# B&R Automation Studio project DeltaTracking
Automation Studio 6.3.0.261; technology packages: mappCockpit 6.0.0, mappMotion 6.4.0, mappView 6.0.0, OpcUaCs 6.0.0

## Configuration Config1

CPU 5APC3100.KBU3-000, AutomationRuntime 6.4.0, Build 11.3.0, Safety 0.0, Vc 

### Task classes (Cpu.sw)
```
Cyclic#1 (cycle 2000 us, tolerance 0 us):
  APP_Convey <- Conveyor.APP_Conveyor1.prg
  APP_Conve1 <- Conveyor.APP_Conveyor2.prg
  APP_Robot1 <- Robots.Robot1.APP_Robot1.prg
DataObjects: Arnc0sys, Acp10sys
NcDataObjects: gmcipuc, gmciplog, gmcipfub, gmcipfun, gmciplsm, gmciplbr, gmcipmxd, gmcipvar, gmcipsys, gmcipiec, gmcipesm, gmcipusm, gmcipcsm, gmcipui, gmcipubr, gmcipcbr, gmcipcfg, gmcipus, gmcipmx, Cam
Binaries: McAcpSys, mcdrivelog, udbdef, TCData, mvLoader, arsvcreg, arflatprv, mCoWebSc, McAcpDrv, McAcpSim, McProfGen, McMechSys, arcoal, ashwac, arconfig, asfw, ashwd, iomap, User, Role, sysconf, TraceConfi, Settings, Config_1, Hierarchy, Config, AxisAx_1, Config_2, ComRobot, Config_4, Config_5, Config_3, Config_6, ToolX20, AxesAxX21, GRobot1, GFRobot1, ARobot1, ComRobot1, WorkRobot1, GRobot2, MRobot1, GFRobot2, FeatX21, TrkDevX21, TrkDevConv, AxisAxX25, MecX20, AxesAxX20, WorkX20, FeatX20, DeltaX20, ComFeatX20, DeltaX21, TrkDevX20, vccddbox, vcfile, vccbtn, vcpdvnc, arialbd, vcmgr, vctcal, vcgclass, vcctext, vccnum, vcfntttf, vcdsloc, vccstr, arial, Visu03, vccshape, vcalarm, Visu01, vccdt, vccscale, vcchtml, vcchspot, vccbmp, vccpopup, vcshared, vcxml, vccurl, vcrt, vccslider, Visu02, vcnet, vcclbox, vcbclass, vcdsint, vcpdsw, vccovl, vccline, TCLang, visvc, vccdbox, vcpfar00, vcpfmtcx, vcpfapc, GrpMaster, Users, UsersLogin, TC, Files, DiagWebXs, AlmMaster, AlmHisMain, AlmMain, GrpVMaster, AlmVMaster, CfgPureVir, AxisPS, AxisAxXX1, AxisAxXX2, AxisMaster, MDevXX1, AxVMaster, GrpDevXX1, AlmDevXX1, GrPDevXX4, AlmDevXX4, GrPDevX10, AlmDevX10, AlmDevX20, GrpDevX20, AlmDevX21, GrpDevX21, AlmMBelts, GrpMBelts, AlmDevXX6, GrpDevXX6, AxesVAxX20, vcpfx20, AxisMBelts, MasMBelts, MBeltsPt, AxesVAxX25, AxesAxX10, AxesAxX25, WorkX10, CncXX6, MecX10, AxesVAxX10, DeltaX10, FeatXX6, FeatX10, ToolX10, ToolXX6, MecXX6, MotMaster, MotVMaster, vcctrend, MotDevX10, GrPDevXX3, AlmDevXX3, MotDevXX3, GrPDevXX2, MotDevXX1, AlmDevXX2, MotDevXX2, vcpkat, arnc0cfg, Sdc10map, Arnc0map, Sdc10map1, Sdc10map2, MotDevX20, MotDevX11, MotDevXX9, GrpDevXX9, AlmDevXX9, PML, MotDevXX6, CncDevXX6, MotDevXX7, AlmDevXX7, GrpDevXX7, Robot, AlmDevXX8, GrpDevXX8, MotSim, MotSpindle, MotDevXXA, AlmDevXXA, GrpDevXXA, GrpDevX11, AlmDevX11, OpcUaBasic, User_1, OpcUaMap, AlmHmi, AlmHistHmi, Groups, vccpiech, MotMac, acp10cfg, Acp10map
Libraries: standard, AsBrStr, sys_lib, runtime, AsArSdm, astime, brsystem, FileIO, AsIODiag, DataObj, AsArProf, AsMem, AsIOAcc, AsEPL, ASMcDcs, AsBrMath, visapi, ArTextSys, AsSem, AsIecCon, AsZip, MpRecipe, MpUserX, MpFile, MpAlarmX, MpCom, CoTrace, MpServer, powerlnk, aruser, asusb, ashw, arcert, arssl, aseth, asio, vcresman, IecCheck, areventlog, MpBase, McBase, McAxGroup, McAcpAx, McAxis, McPathGen, McTrkPath, MpAxis, McProgInt, McPureVAx, McDS402Ax, MpRobotics, MpCnc
```

### Hardware
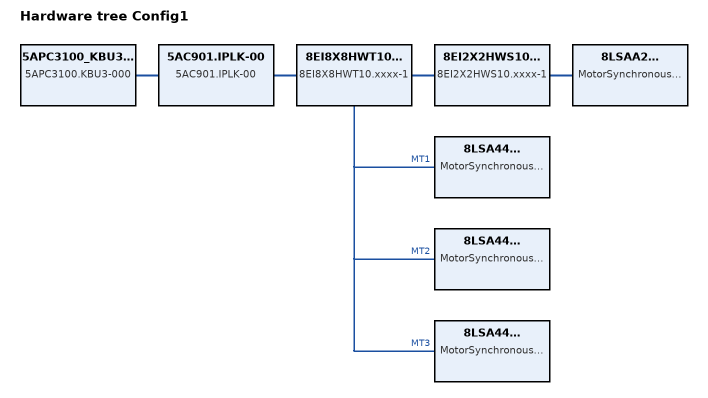
```
5AC901.IPLK-00 : 5AC901.IPLK-00 v2.0.0.0  [SL -> 5APC3100_KBU3_000.SL2]
  Connector IF1:
    DNAConfiguration = manual
    Channel1
    ChannelID1 = McAcpBroadcast
    ChannelType1 = OCTET[96]
5APC3100_KBU3_000 : 5APC3100.KBU3-000 v2.2.7.0
  Connector IF3:
    AssignedOperatingSystem = ARemb
    ActivateDevice = 1
    HostName = apc3100robert
    Mode = Manual
    InternetAddress = 10.43.51.43
    SubnetMask = 255.255.255.0
    Vnc1
    VncKeyMappingFile1 = 
    VncRefreshRate1 = 100
    ActivateSnmp = 2
  Connector IF4:
    AssignedOperatingSystem = ARemb
    ActivateDevice = 1
    HostName = apc3100robert
    Mode = DHCPServer
    InternetAddress = 192.168.20.254
    SubnetMask = 255.255.255.0
    Lease1
    LeaseName1 = Range1
    LeaseStartAddress1 = 192.168.20.100
    LeaseStopAddress1 = 192.168.20.110
    LeaseSubnetMask1 = 255.255.255.0
    Vnc1
    VncTitle1 = VNC
    ActivateSnmp = 2
  Connector IF5:
    AssignedOperatingSystem = ARemb
  Connector IF6:
    AssignedOperatingSystem = ARemb
  Connector IF7:
    AssignedOperatingSystem = ARemb
  Connector IF8:
    AssignedOperatingSystem = ARemb
  ConfigurationID = Template_X20CP1586
  UserPartitionSize = 5
  Simulation = 1
  TimerDeviceType = EPLX2X
  TimerDevice = 5AC901.IPLK-00.IF1
  IdleTaskClass = 4
  TaskClassIdleTime = 4000
  Cyclic1Duration = 2000
  Cyclic1Tolerance = 0
  Cyclic1Stack = 16384
  Cyclic2Duration = 4000
  Cyclic2Tolerance = 0
  Cyclic3Duration = 10000
  Cyclic3Tolerance = 0
  Cyclic4Duration = 20000
  Cyclic4Tolerance = 0
  Cyclic5Duration = 50000
  Cyclic5Tolerance = 0
  Cyclic6Duration = 100000
  Cyclic6Tolerance = 0
  Cyclic7Duration = 200000
  Cyclic7Tolerance = 0
  FileDevice1
  FileDeviceName1 = SceneViewer
  FileDevicePath1 = USER_PATH
  FileDevice2
  FileDeviceName2 = MPLogDir
  FileDevicePath2 = USER_PATH\Log
  FileDevice3
  FileDeviceName3 = DebugData
  FileDevicePath3 = USER_PATH\\Debug
  FileDevice4
  FileDeviceName4 = CNC_Prg
  FileDevicePath4 = USER_PATH\CNC_Prg
  EthernetDefaultGateway = 10.43.51.1
  ActivateFtpServer = 1
  FTPProtocol = 2
  FtpUser1
  FtpUsername1 = gmctest
  FtpUserPassword1 = dJg12F/7hd2fGO/QauVo5qNTeUud8LRwkPqca2btE1Q=
  FtpUserSalt1 = iGhlfz5v
  FTPAccessRight1 = 0
  FTPdevice1 = ALL
  ActivateWebServer = 1
  ActivateSdm = 1
8EI2X2HWS10.xxxx-1-QC_D4r1100R_1 : 8EI2X2HWS10.xxxx-1 v2.4.0.0 (NodeNumber=6)  [PLK1 -> 8EI8X8HWT10.xxxx-1-Q1-Q2-Q3_D4r1100R_1.PLK2 [Cable Type=PowerlinkCable, Length=10, Version=1.0.0.3]]
  DriveConfiguration/Encoder/EncoderX41:
    InterfaceType = EnDat
  DriveConfiguration/Channel[1]/RealAxis:
    AxisReference = gAxisQC_D4r1100R_1
  DriveConfiguration/Channel[1]/RealAxis/MechanicalElements/Gearbox:
    InputIsReadOnly = 1
    Input = 10
    OutputIsReadOnly = 1
  DriveConfiguration/Channel[1]/RealAxis/MechanicalElements/RotaryToLinearTransformation:
    ReferenceDistanceIsReadOnly = 1
    ReferenceDistance = 360
  DriveConfiguration/Channel[1]/RealAxis/Controller:
    ModeIsReadOnly = 1
    Mode = PositionControllerWithTorqueFeedForward
  DriveConfiguration/Channel[1]/RealAxis/Controller/Mode/Position:
    ProportionalGainIsReadOnly = 1
    ProportionalGain = 80.0
    IntegrationTimeIsReadOnly = 1
  DriveConfiguration/Channel[1]/RealAxis/Controller/Mode/Speed:
    ProportionalGainIsReadOnly = 1
    IntegrationTimeIsReadOnly = 1
    FilterTimeIsReadOnly = 1
  DriveConfiguration/Channel[1]/RealAxis/Controller/Mode:
    FeedForwardIsReadOnly = 1
    FeedForward = CyclicValueFromAxesGroup
  DriveConfiguration/Channel[1]/RealAxis/Controller/Mode/LoopFilters:
    LoopFilterXIsReadOnly = 1
  DriveConfiguration/Channel[1]/RealAxis/Homing:
    Mode = Absolute
    RestorePositionVariable = 
  DriveConfiguration/Channel[1]/RealAxis/StopReaction:
    DriveError = CyclicDecelerationFromAxesGroup
  DriveConfiguration/Channel[1]/RealAxis/MovementErrorLimits:
    PositionError = 0.5
  DriveConfiguration/Channel[1]/RealAxis:
    JerkFilterIsReadOnly = 1
    JerkFilter = Used
  DriveConfiguration/Channel[1]/RealAxis/JerkFilter:
    JerkTimeMin = 0.06
    JerkTime = 0.06
8EI8X8HWT10.xxxx-1-Q1-Q2-Q3_D4r1100R_1 : 8EI8X8HWT10.xxxx-1 v2.4.0.0 (NodeNumber=4)  [PLK1 -> 5AC901.IPLK-00.IF1 [Cable Type=PowerlinkCable, Length=10, Version=1.0.0.3]; PLK2 -> 8EI2X2HWS10.xxxx-1-QC_D4r1100R_1.PLK1 [Cable Type=PowerlinkCable, Length=10, Version=1.0.0.3]; MT2 -> 8LSA44.DB060S200-3_Q2_D4r1100R_1.MT; MT3 -> 8LSA44.DB060S200-3_Q3_D4r1100R_1.MT]
  DriveConfiguration/Encoder/EncoderX41:
    InterfaceType = EnDat
  DriveConfiguration/Encoder/EncoderX42:
    InterfaceType = EnDat
  DriveConfiguration/Encoder/EncoderX43:
    InterfaceType = EnDat
  DriveConfiguration/Channel[1]/RealAxis:
    AxisReference = gAxisQ1_D4r1100R_1
  DriveConfiguration/Channel[1]/RealAxis/MechanicalElements/Gearbox:
    InputIsReadOnly = 1
    Input = 28
    OutputIsReadOnly = 1
  DriveConfiguration/Channel[1]/RealAxis/MechanicalElements/RotaryToLinearTransformation:
    ReferenceDistanceIsReadOnly = 1
    ReferenceDistance = 360
  DriveConfiguration/Channel[1]/RealAxis/Controller:
    ModeIsReadOnly = 1
    Mode = PositionControllerWithTorqueFeedForward
  DriveConfiguration/Channel[1]/RealAxis/Controller/Mode/Position:
    ProportionalGainIsReadOnly = 1
    ProportionalGain = 150.0
    IntegrationTimeIsReadOnly = 1
  DriveConfiguration/Channel[1]/RealAxis/Controller/Mode/Speed:
    ProportionalGainIsReadOnly = 1
    ProportionalGain = 7.5
    IntegrationTimeIsReadOnly = 1
    FilterTimeIsReadOnly = 1
  DriveConfiguration/Channel[1]/RealAxis/Controller/Mode:
    FeedForwardIsReadOnly = 1
    FeedForward = CyclicValueFromAxesGroup
  DriveConfiguration/Channel[1]/RealAxis/Controller/Mode/LoopFilters:
    LoopFilterXIsReadOnly = 1
  DriveConfiguration/Channel[1]/RealAxis/Homing:
    Mode = Absolute
    RestorePositionVariable = 
  DriveConfiguration/Channel[1]/RealAxis/StopReaction:
    DriveError = CyclicDecelerationFromAxesGroup
  DriveConfiguration/Channel[1]/RealAxis/MovementErrorLimits:
    PositionError = 0.5
  DriveConfiguration/Channel[1]/RealAxis:
    JerkFilterIsReadOnly = 1
    JerkFilter = Used
  DriveConfiguration/Channel[1]/RealAxis/JerkFilter:
    JerkTimeMin = 0.06
    JerkTime = 0.06
  DriveConfiguration/Channel[2]/RealAxis:
    AxisReference = gAxisQ2_D4r1100R_1
  DriveConfiguration/Channel[2]/RealAxis/MechanicalElements/Gearbox:
    InputIsReadOnly = 1
    Input = 28
    OutputIsReadOnly = 1
  DriveConfiguration/Channel[2]/RealAxis/MechanicalElements/RotaryToLinearTransformation:
    ReferenceDistanceIsReadOnly = 1
    ReferenceDistance = 360
  DriveConfiguration/Channel[2]/RealAxis/Controller:
    ModeIsReadOnly = 1
    Mode = PositionControllerWithTorqueFeedForward
  DriveConfiguration/Channel[2]/RealAxis/Controller/Mode/Position:
    ProportionalGainIsReadOnly = 1
    ProportionalGain = 150.0
    IntegrationTimeIsReadOnly = 1
  DriveConfiguration/Channel[2]/RealAxis/Controller/Mode/Speed:
    ProportionalGainIsReadOnly = 1
    ProportionalGain = 7.5
    IntegrationTimeIsReadOnly = 1
    FilterTimeIsReadOnly = 1
  DriveConfiguration/Channel[2]/RealAxis/Controller/Mode:
    FeedForwardIsReadOnly = 1
    FeedForward = CyclicValueFromAxesGroup
  DriveConfiguration/Channel[2]/RealAxis/Controller/Mode/LoopFilters:
    LoopFilterXIsReadOnly = 1
  DriveConfiguration/Channel[2]/RealAxis/Homing:
    Mode = Absolute
    RestorePositionVariable = 
  DriveConfiguration/Channel[2]/RealAxis/StopReaction:
    DriveError = CyclicDecelerationFromAxesGroup
  DriveConfiguration/Channel[2]/RealAxis/MovementErrorLimits:
    PositionError = 0.5
  DriveConfiguration/Channel[2]/RealAxis:
    JerkFilterIsReadOnly = 1
    JerkFilter = Used
  DriveConfiguration/Channel[2]/RealAxis/JerkFilter:
    JerkTimeMin = 0.06
    JerkTime = 0.06
  DriveConfiguration/Channel[3]/RealAxis:
    AxisReference = gAxisQ3_D4r1100R_1
  DriveConfiguration/Channel[3]/RealAxis/MechanicalElements/Gearbox:
    InputIsReadOnly = 1
    Input = 28
    OutputIsReadOnly = 1
  DriveConfiguration/Channel[3]/RealAxis/MechanicalElements/RotaryToLinearTransformation:
    ReferenceDistanceIsReadOnly = 1
    ReferenceDistance = 360
  DriveConfiguration/Channel[3]/RealAxis/Controller:
    ModeIsReadOnly = 1
    Mode = PositionControllerWithTorqueFeedForward
  DriveConfiguration/Channel[3]/RealAxis/Controller/Mode/Position:
    ProportionalGainIsReadOnly = 1
    ProportionalGain = 150.0
    IntegrationTimeIsReadOnly = 1
  DriveConfiguration/Channel[3]/RealAxis/Controller/Mode/Speed:
    ProportionalGainIsReadOnly = 1
    ProportionalGain = 7.5
    IntegrationTimeIsReadOnly = 1
    FilterTimeIsReadOnly = 1
  DriveConfiguration/Channel[3]/RealAxis/Controller/Mode:
    FeedForwardIsReadOnly = 1
    FeedForward = CyclicValueFromAxesGroup
  DriveConfiguration/Channel[3]/RealAxis/Controller/Mode/LoopFilters:
    LoopFilterXIsReadOnly = 1
  DriveConfiguration/Channel[3]/RealAxis/Homing:
    Mode = Absolute
    RestorePositionVariable = 
  DriveConfiguration/Channel[3]/RealAxis/StopReaction:
    DriveError = CyclicDecelerationFromAxesGroup
  DriveConfiguration/Channel[3]/RealAxis/MovementErrorLimits:
    PositionError = 0.5
  DriveConfiguration/Channel[3]/RealAxis:
    JerkFilterIsReadOnly = 1
    JerkFilter = Used
  DriveConfiguration/Channel[3]/RealAxis/JerkFilter:
    JerkTimeMin = 0.06
    JerkTime = 0.06
8LSA44.DB060S200-3_Q1_D4r1100R_1 : MotorSynchronous_any v2.2.1.0  [MT -> 8EI8X8HWT10.xxxx-1-Q1-Q2-Q3_D4r1100R_1.MT1]
  M1/MotorParameters:
    MOTOR_POLEPAIRS = 5
    MOTOR_SPEED_RATED = 6000
    MOTOR_SPEED_MAX = 12000
    MOTOR_VOLTAGE_RATED = 400
    MOTOR_CURR_RATED = 3.7
    MOTOR_CURR_STALL = 7.4
    MOTOR_CURR_MAX = 43.8
    MOTOR_TORQ_RATED = 3
    MOTOR_TORQ_STALL = 6
    MOTOR_TORQ_MAX = 22.8
    MOTOR_VOLTAGE_CONST = 49.22
    MOTOR_TORQ_CONST = 0.81
    MOTOR_STATOR_RESISTANCE = 0.863
    MOTOR_STATOR_INDUCTANCE = 6.2
    MOTOR_INERTIA = 2.73
    VoltageLimitation = Used
  M1/MotorParameters/VoltageLimitation:
    MOTOR_UDC_MAX = 1000
  M1/MotorParameters/EncoderMounting:
    Angle = StoredOnEncoder
  M1/MotorParameters/TemperatureSensor:
    MOTOR_TEMPSENS_LIM = 130
    TemperatureSensorInterface = EncoderConnectorDigital
    MOTOR_TEMPSENS_PAR1 = 30
    MOTOR_TEMPSENS_PAR2 = 254
    MOTOR_TEMPSENS_PAR3 = -29.72
    MOTOR_TEMPSENS_PAR4 = -4.58
    MOTOR_TEMPSENS_PAR5 = 20.33
    MOTOR_TEMPSENS_PAR6 = 45.18
    MOTOR_TEMPSENS_PAR7 = 69.96
    MOTOR_TEMPSENS_PAR8 = 94.71
    MOTOR_TEMPSENS_PAR9 = 119.6
    MOTOR_TEMPSENS_PAR10 = 149.11
  M1/MotorParameters/TemperatureModel:
    MOTOR_WIND_TEMP_MAX = 110
  M1/MotorParameters/TemperatureModel/Calculation:
    MOTOR_WIND_CROSS_SECT = 0.985
    MOTOR_TAU_THERM = 1800
  M1:
    Brake = Used
  M1/Brake:
    MOTOR_BRAKE_CURR_RATED = 0.83
    MOTOR_BRAKE_TORQ_RATED = 8
    MOTOR_BRAKE_ON_TIME = 0.038
    MOTOR_BRAKE_OFF_TIME = 0.055
    MOTOR_BRAKE_INERTIA = 0.69
  M1/Encoder:
    MOTOR_ENCOD_ATTR = 1
    MOTOR_ENCOD_INERTIA = 0.022
    TemperatureSensor = Used
  M1/Encoder/TemperatureSensor:
    MOTOR_ENCOD_TEMP_LIM = 129
  M1:
    Gearbox = UsedWithDynamicTorqueLimitation
  M1/Gearbox/GearRatio:
    Input = 28
  M1/Gearbox:
    MOTORGEAR_SPEED_MAX = 7500
    MOTORGEAR_TORQ_NOM = 126
    MOTORGEAR_TORQ_MAX = 126
    MOTORGEAR_INERTIA = 0.51
    MOTORGEAR_VISC_FRIC = 0.002
    MOTORGEAR_STAT_FRIC = 0.22
8LSA44.DB060S200-3_Q2_D4r1100R_1 : MotorSynchronous_any v2.2.1.0  [MT -> 8EI8X8HWT10.xxxx-1-Q1-Q2-Q3_D4r1100R_1.MT2]
  M1/MotorParameters:
    MOTOR_POLEPAIRS = 5
    MOTOR_SPEED_RATED = 6000
    MOTOR_SPEED_MAX = 12000
    MOTOR_VOLTAGE_RATED = 400
    MOTOR_CURR_RATED = 3.7
    MOTOR_CURR_STALL = 7.4
    MOTOR_CURR_MAX = 43.8
    MOTOR_TORQ_RATED = 3
    MOTOR_TORQ_STALL = 6
    MOTOR_TORQ_MAX = 22.8
    MOTOR_VOLTAGE_CONST = 49.22
    MOTOR_TORQ_CONST = 0.81
    MOTOR_STATOR_RESISTANCE = 0.863
    MOTOR_STATOR_INDUCTANCE = 6.2
    MOTOR_INERTIA = 2.73
    VoltageLimitation = Used
  M1/MotorParameters/VoltageLimitation:
    MOTOR_UDC_MAX = 1000
  M1/MotorParameters/EncoderMounting:
    Angle = StoredOnEncoder
  M1/MotorParameters/TemperatureSensor:
    MOTOR_TEMPSENS_LIM = 130
    TemperatureSensorInterface = EncoderConnectorDigital
    MOTOR_TEMPSENS_PAR1 = 30
    MOTOR_TEMPSENS_PAR2 = 254
    MOTOR_TEMPSENS_PAR3 = -29.72
    MOTOR_TEMPSENS_PAR4 = -4.58
    MOTOR_TEMPSENS_PAR5 = 20.33
    MOTOR_TEMPSENS_PAR6 = 45.18
    MOTOR_TEMPSENS_PAR7 = 69.96
    MOTOR_TEMPSENS_PAR8 = 94.71
    MOTOR_TEMPSENS_PAR9 = 119.6
    MOTOR_TEMPSENS_PAR10 = 149.11
  M1/MotorParameters/TemperatureModel:
    MOTOR_WIND_TEMP_MAX = 110
  M1/MotorParameters/TemperatureModel/Calculation:
    MOTOR_WIND_CROSS_SECT = 0.985
    MOTOR_TAU_THERM = 1800
  M1:
    Brake = Used
  M1/Brake:
    MOTOR_BRAKE_CURR_RATED = 0.83
    MOTOR_BRAKE_TORQ_RATED = 8
    MOTOR_BRAKE_ON_TIME = 0.038
    MOTOR_BRAKE_OFF_TIME = 0.055
    MOTOR_BRAKE_INERTIA = 0.69
  M1/Encoder:
    MOTOR_ENCOD_ATTR = 1
    MOTOR_ENCOD_INERTIA = 0.022
    TemperatureSensor = Used
  M1/Encoder/TemperatureSensor:
    MOTOR_ENCOD_TEMP_LIM = 129
  M1:
    Gearbox = UsedWithDynamicTorqueLimitation
  M1/Gearbox/GearRatio:
    Input = 28
  M1/Gearbox:
    MOTORGEAR_SPEED_MAX = 7500
    MOTORGEAR_TORQ_NOM = 126
    MOTORGEAR_TORQ_MAX = 126
    MOTORGEAR_INERTIA = 0.51
    MOTORGEAR_VISC_FRIC = 0.002
    MOTORGEAR_STAT_FRIC = 0.22
8LSA44.DB060S200-3_Q3_D4r1100R_1 : MotorSynchronous_any v2.2.1.0  [MT -> 8EI8X8HWT10.xxxx-1-Q1-Q2-Q3_D4r1100R_1.MT3]
  M1/MotorParameters:
    MOTOR_POLEPAIRS = 5
    MOTOR_SPEED_RATED = 6000
    MOTOR_SPEED_MAX = 12000
    MOTOR_VOLTAGE_RATED = 400
    MOTOR_CURR_RATED = 3.7
    MOTOR_CURR_STALL = 7.4
    MOTOR_CURR_MAX = 43.8
    MOTOR_TORQ_RATED = 3
    MOTOR_TORQ_STALL = 6
    MOTOR_TORQ_MAX = 22.8
    MOTOR_VOLTAGE_CONST = 49.22
    MOTOR_TORQ_CONST = 0.81
    MOTOR_STATOR_RESISTANCE = 0.863
    MOTOR_STATOR_INDUCTANCE = 6.2
    MOTOR_INERTIA = 2.73
    VoltageLimitation = Used
  M1/MotorParameters/VoltageLimitation:
    MOTOR_UDC_MAX = 1000
  M1/MotorParameters/EncoderMounting:
    Angle = StoredOnEncoder
  M1/MotorParameters/TemperatureSensor:
    MOTOR_TEMPSENS_LIM = 130
    TemperatureSensorInterface = EncoderConnectorDigital
    MOTOR_TEMPSENS_PAR1 = 30
    MOTOR_TEMPSENS_PAR2 = 254
    MOTOR_TEMPSENS_PAR3 = -29.72
    MOTOR_TEMPSENS_PAR4 = -4.58
    MOTOR_TEMPSENS_PAR5 = 20.33
    MOTOR_TEMPSENS_PAR6 = 45.18
    MOTOR_TEMPSENS_PAR7 = 69.96
    MOTOR_TEMPSENS_PAR8 = 94.71
    MOTOR_TEMPSENS_PAR9 = 119.6
    MOTOR_TEMPSENS_PAR10 = 149.11
  M1/MotorParameters/TemperatureModel:
    MOTOR_WIND_TEMP_MAX = 110
  M1/MotorParameters/TemperatureModel/Calculation:
    MOTOR_WIND_CROSS_SECT = 0.985
    MOTOR_TAU_THERM = 1800
  M1:
    Brake = Used
  M1/Brake:
    MOTOR_BRAKE_CURR_RATED = 0.83
    MOTOR_BRAKE_TORQ_RATED = 8
    MOTOR_BRAKE_ON_TIME = 0.038
    MOTOR_BRAKE_OFF_TIME = 0.055
    MOTOR_BRAKE_INERTIA = 0.69
  M1/Encoder:
    MOTOR_ENCOD_ATTR = 1
    MOTOR_ENCOD_INERTIA = 0.022
    TemperatureSensor = Used
  M1/Encoder/TemperatureSensor:
    MOTOR_ENCOD_TEMP_LIM = 129
  M1:
    Gearbox = UsedWithDynamicTorqueLimitation
  M1/Gearbox/GearRatio:
    Input = 28
  M1/Gearbox:
    MOTORGEAR_SPEED_MAX = 7500
    MOTORGEAR_TORQ_NOM = 126
    MOTORGEAR_TORQ_MAX = 126
    MOTORGEAR_INERTIA = 0.51
    MOTORGEAR_VISC_FRIC = 0.002
    MOTORGEAR_STAT_FRIC = 0.22
8LSAA2.D9045S200-3_QC_D4r1100R_1 : MotorSynchronous_any v2.2.1.0  [MT -> 8EI2X2HWS10.xxxx-1-QC_D4r1100R_1.MT1]
  M1/MotorParameters:
    MOTOR_POLEPAIRS = 5
    MOTOR_SPEED_RATED = 4500
    MOTOR_SPEED_MAX = 7000
    MOTOR_VOLTAGE_RATED = 400
    MOTOR_CURR_RATED = 1.31
    MOTOR_CURR_STALL = 1.42
    MOTOR_CURR_MAX = 6
    MOTOR_TORQ_RATED = 1.27
    MOTOR_TORQ_STALL = 1.4
    MOTOR_TORQ_MAX = 4.5
    MOTOR_VOLTAGE_CONST = 58.64
    MOTOR_TORQ_CONST = 0.97
    MOTOR_STATOR_RESISTANCE = 13.9
    MOTOR_STATOR_INDUCTANCE = 27
    MOTOR_INERTIA = 0.38
    VoltageLimitation = Used
  M1/MotorParameters/VoltageLimitation:
    MOTOR_UDC_MAX = 1000
  M1/MotorParameters/EncoderMounting:
    Angle = StoredOnEncoder
  M1/MotorParameters/TemperatureSensor:
    MOTOR_TEMPSENS_LIM = 130
    TemperatureSensorInterface = EncoderConnectorDigital
    MOTOR_TEMPSENS_PAR1 = 30
    MOTOR_TEMPSENS_PAR2 = 254
    MOTOR_TEMPSENS_PAR3 = -29.72
    MOTOR_TEMPSENS_PAR4 = -4.58
    MOTOR_TEMPSENS_PAR5 = 20.33
    MOTOR_TEMPSENS_PAR6 = 45.18
    MOTOR_TEMPSENS_PAR7 = 69.96
    MOTOR_TEMPSENS_PAR8 = 94.71
    MOTOR_TEMPSENS_PAR9 = 119.6
    MOTOR_TEMPSENS_PAR10 = 149.11
  M1/MotorParameters/TemperatureModel:
    MOTOR_WIND_TEMP_MAX = 110
  M1/MotorParameters/TemperatureModel/Calculation:
    MOTOR_WIND_CROSS_SECT = 0.126
    MOTOR_TAU_THERM = 1860
  M1:
    Brake = Used
  M1/Brake:
    MOTOR_BRAKE_CURR_RATED = 0.56
    MOTOR_BRAKE_TORQ_RATED = 3.2
    MOTOR_BRAKE_ON_TIME = 0.01
    MOTOR_BRAKE_OFF_TIME = 0.06
    MOTOR_BRAKE_INERTIA = 0.38
  M1/Encoder:
    MOTOR_ENCOD_ATTR = 1
    MOTOR_ENCOD_INERTIA = 0.004
    TemperatureSensor = Used
  M1/Encoder/TemperatureSensor:
    MOTOR_ENCOD_TEMP_LIM = 124
  M1:
    Gearbox = UsedWithDynamicTorqueLimitation
  M1/Gearbox/GearRatio:
    Input = 10
  M1/Gearbox:
    MOTORGEAR_SPEED_MAX = 7500
    MOTORGEAR_TORQ_NOM = 7.0
    MOTORGEAR_TORQ_MAX = 7.0
    MOTORGEAR_INERTIA = 0.16
    MOTORGEAR_VISC_FRIC = 0.0038
    MOTORGEAR_STAT_FRIC = 0.07
```

### Config_11.axesgroupfeature - 5APC3100_KBU3_000/mappMotion/Codian_D4r1100R_1/Config_11.axesgroupfeature
```
Element Feature_Programs_D4r1100R_1 (Type=axesgroupfeature)
  Type:
    InitialSettings:
      AccuracyHoldDelays = User defined
        UserAxesDelay = 0.03
    Location = User
      UserLocation[1]:
        FileDevice = CNC_Prg
```

### Config_2.axesgroup - 5APC3100_KBU3_000/mappMotion/Codian_D4r1100R_1/Config_2.axesgroup
```
Element gAxesGroup_D4r1100R_1 (Type=axesgroup)
  Type = PathGenAxesGroup
    ProcessingTaskClass = 1
    License = 1
    PhysicalAxes:
      JointAxes:
        JointAxisAxisRefIsReadOnly = 0
        JointAxis[1]:
          Name = Q1
          AxisRef = gAxisQ1_D4r1100R_1
        JointAxis[2]:
          Name = Q2
          AxisRef = gAxisQ2_D4r1100R_1
        JointAxis[3]:
          Name = Q3
          AxisRef = gAxisQ3_D4r1100R_1
        JointAxis[4]:
          Name = QC
          AxisRef = gAxisQC_D4r1100R_1
    MechanicalSystem:
      MechSysRefIsReadOnly = 0
      MechSysRef = MechSys_D4r1100R_1
    BasicSettings:
      ModalDataBehaviour = ResetToDefault
      GeometryPlanning:
        TCPResolutionIsReadOnly = 0
        TCPResolution:
          LengthResolution = 0.001
          AngleResolution = 0.001
        Rounding:
          PathDistance = 0.0
          SymmetricRounding = Yes
          LastSegment = Half
          AvoidZeroCurvature = No
        RoundingMode = Standard
        MaxCornerDeviation = 0.0
        MaxTangentialTransitionDeviation = 0.05
        MaxRadiusDeviation = 0.001
        WorkingPlane = XY
      TrajectoryPlanningIsReadOnly = 0
      TrajectoryPlanning = Basic
        LimitCheckResolutionIsReadOnly = 0
        LimitCheckResolution = UserDefinedTime
          TimeIsReadOnly = 0
          Time = 0.005
        BufferTime = UserDefinedTime
          Time = 0.05
        BarrierParametrization = JointCoordinates
        TorqueLimitConsideration = Exact
      Miscellaneous:
        NonMovementsLimit = NotUsed
        TimeStretchOverride:
          JerkSuppression = NotUsed
    StopReaction:
      AxisError:
        AxisReactionIsReadOnly = 0
    AxesGroupFeatures:
      FeatureRef[1] = Feature_Programs_D4r1100R_1
      FeatureRef[2] = Feature_FrameHierachy
      FeatureRef[3] = Feature_InterpreterLog
      FeatureRef[4] = Feature_MFunctions
      FeatureRef[5] = Feature_Monitoring
      FeatureRef[6] = Feature_PathDefRobot
      FeatureRef[7] = Feature_TrackingRobot
    SceneObject:
      FileDevice = ComponentScenes
      FileNamePrefix = PathGen_
      FrameSize = 150
      FrameName = Invisible
      Positioner = NotUsed
      Object = Visible
      Boundaries = NotUsed
  Alarms = None
```

### Config_3.axis - 5APC3100_KBU3_000/mappMotion/Codian_D4r1100R_1/Config_3.axis
```
Element gAxisQ1_D4r1100R_1 (Type=axis)
  BaseTypeIsReadOnly = 1
  BaseType = RotaryBounded
    MeasurementUnitIsReadOnly = 1
    MeasurementUnit = 17476
    MeasurementResolutionIsReadOnly = 1
    MeasurementResolution = 0.001
    CountDirectionIsReadOnly = 1
    CountDirection = Inverse
  MovementLimitsIsReadOnly = 1
  MovementLimits = InternalForPathControlledAxis
    Position:
      LowerLimitMin = -47
      UpperLimitMax = 99.5
      LowerLimit = -47
      UpperLimit = 99.5
    VelocityIsReadOnly = 1
    Velocity:
      VelocityMax = 1160
      Velocity = 1160
    AccelerationIsReadOnly = 1
    Acceleration:
      AccelerationMax = 35000
      Acceleration = 35000
    DecelerationIsReadOnly = 1
    Deceleration:
      DecelerationMax = 35000
      Deceleration = 35000
    JerkIsReadOnly = 1
    Jerk = Advanced
      JerkAccelerationPositiveMin = 0
      JerkAccelerationPositiveMax = 2200000
      JerkAccelerationPositive = 2200000
      JerkAccelerationNegativeMin = 0
      JerkAccelerationNegativeMax = 2200000
      JerkAccelerationNegative = 2200000
      JerkDecelerationPositiveMin = 0
      JerkDecelerationPositiveMax = 2000000
      JerkDecelerationPositive = 2000000
      JerkDecelerationNegativeMin = 0
      JerkDecelerationNegativeMax = 2000000
      JerkDecelerationNegative = 2000000
    TorqueIsInvisible = 0
    TorqueIsReadOnly = 1
    Torque = Basic
      TorqueMax = 20.5
      Torque = 20.5
  Alarms = None
Element gAxisQ2_D4r1100R_1 (Type=axis)
  BaseTypeIsReadOnly = 1
  BaseType = RotaryBounded
    MeasurementUnitIsReadOnly = 1
    MeasurementUnit = 17476
    MeasurementResolutionIsReadOnly = 1
    MeasurementResolution = 0.001
    CountDirectionIsReadOnly = 1
    CountDirection = Inverse
  MovementLimitsIsReadOnly = 1
  MovementLimits = InternalForPathControlledAxis
    Position:
      LowerLimitMin = -47
      UpperLimitMax = 99.5
      LowerLimit = -47
      UpperLimit = 99.5
    VelocityIsReadOnly = 1
    Velocity:
      VelocityMax = 1160
      Velocity = 1160
    AccelerationIsReadOnly = 1
    Acceleration:
      AccelerationMax = 35000
      Acceleration = 35000
    DecelerationIsReadOnly = 1
    Deceleration:
      DecelerationMax = 35000
      Deceleration = 35000
    JerkIsReadOnly = 1
    Jerk = Advanced
      JerkAccelerationPositiveMin = 0
      JerkAccelerationPositiveMax = 2200000
      JerkAccelerationPositive = 2200000
      JerkAccelerationNegativeMin = 0
      JerkAccelerationNegativeMax = 2200000
      JerkAccelerationNegative = 2200000
      JerkDecelerationPositiveMin = 0
      JerkDecelerationPositiveMax = 2000000
      JerkDecelerationPositive = 2000000
      JerkDecelerationNegativeMin = 0
      JerkDecelerationNegativeMax = 2000000
      JerkDecelerationNegative = 2000000
    TorqueIsInvisible = 0
    TorqueIsReadOnly = 1
    Torque = Basic
      TorqueMax = 20.5
      Torque = 20.5
  Alarms = None
Element gAxisQ3_D4r1100R_1 (Type=axis)
  BaseTypeIsReadOnly = 1
  BaseType = RotaryBounded
    MeasurementUnitIsReadOnly = 1
    MeasurementUnit = 17476
    MeasurementResolutionIsReadOnly = 1
    MeasurementResolution = 0.001
    CountDirectionIsReadOnly = 1
    CountDirection = Inverse
  MovementLimitsIsReadOnly = 1
  MovementLimits = InternalForPathControlledAxis
    Position:
      LowerLimitMin = -47
      UpperLimitMax = 99.5
      LowerLimit = -47
      UpperLimit = 99.5
    VelocityIsReadOnly = 1
    Velocity:
      VelocityMax = 1160
      Velocity = 1160
    AccelerationIsReadOnly = 1
    Acceleration:
      AccelerationMax = 35000
      Acceleration = 35000
    DecelerationIsReadOnly = 1
    Deceleration:
      DecelerationMax = 35000
      Deceleration = 35000
    JerkIsReadOnly = 1
    Jerk = Advanced
      JerkAccelerationPositiveMin = 0
      JerkAccelerationPositiveMax = 2200000
      JerkAccelerationPositive = 2200000
      JerkAccelerationNegativeMin = 0
      JerkAccelerationNegativeMax = 2200000
      JerkAccelerationNegative = 2200000
      JerkDecelerationPositiveMin = 0
      JerkDecelerationPositiveMax = 2000000
      JerkDecelerationPositive = 2000000
      JerkDecelerationNegativeMin = 0
      JerkDecelerationNegativeMax = 2000000
      JerkDecelerationNegative = 2000000
    TorqueIsInvisible = 0
    TorqueIsReadOnly = 1
    Torque = Basic
      TorqueMax = 20.5
      Torque = 20.5
  Alarms = None
Element gAxisQC_D4r1100R_1 (Type=axis)
  BaseTypeIsReadOnly = 1
  BaseType = Rotary
    MeasurementUnitIsReadOnly = 1
    MeasurementUnit = 17476
    MeasurementResolutionIsReadOnly = 1
    MeasurementResolution = 0.001
    CountDirectionIsReadOnly = 1
    CountDirection = Standard
  MovementLimitsIsReadOnly = 1
  MovementLimits = InternalForPathControlledAxis
    Position:
      LowerLimitMin = -1000.0
      UpperLimitMax = 1000.0
      LowerLimit = -1000.0
      UpperLimit = 1000.0
    VelocityIsReadOnly = 1
    Velocity:
      VelocityMax = 3600
      Velocity = 3600
    AccelerationIsReadOnly = 1
    Acceleration:
      AccelerationMax = 50000
      Acceleration = 50000
    DecelerationIsReadOnly = 1
    Deceleration:
      DecelerationMax = 50000
      Deceleration = 50000
    JerkIsReadOnly = 1
    Jerk = Advanced
      JerkAccelerationPositiveMin = 0
      JerkAccelerationPositiveMax = 10000000
      JerkAccelerationPositive = 10000000
      JerkAccelerationNegativeMin = 0
      JerkAccelerationNegativeMax = 10000000
      JerkAccelerationNegative = 10000000
      JerkDecelerationPositiveMin = 0
      JerkDecelerationPositiveMax = 10000000
      JerkDecelerationPositive = 10000000
      JerkDecelerationNegativeMin = 0
      JerkDecelerationNegativeMax = 10000000
      JerkDecelerationNegative = 10000000
    TorqueIsInvisible = 0
    TorqueIsReadOnly = 1
    Torque = Basic
      TorqueMax = 4.0
      Torque = 4.0
  Alarms = None
```

### Config_4.mechanicalsystem - 5APC3100_KBU3_000/mappMotion/Codian_D4r1100R_1/Config_4.mechanicalsystem
```
Element MechSys_D4r1100R_1 (Type=mechanicalsystem)
  TypeIsReadOnly = 1
  Type = Delta
    SubtypeIsReadOnly = 1
    Subtype = 4AxesDeltaA
      SceneViewerObject = Generic
      DescriptionIsReadOnly = 1
      Description = Standard
        Dimensions:
          BasePlatform:
            CenterIsReadOnly = 0
            Center:
              X = 0.0
              Y = 0.0
              Z = 0
            ArmLinkPointIsReadOnly = 0
            Arm1LinkPoint:
              Angle = 0.0
              Radius = 200
              Z = -90
            Arm2LinkPoint:
              Angle = -120.0
              Radius = 200
              Z = -90
            Arm3LinkPoint:
              Angle = -240.0
              Radius = 200
              Z = -90
          Arms:
            ArmIsReadOnly = 0
            Arm1:
              UpperArmLength = 320
              LowerArmLength = 850
            Arm2:
              UpperArmLength = 320
              LowerArmLength = 850
            Arm3:
              UpperArmLength = 320
              LowerArmLength = 850
            LowerArmPairDistance = 105
          EndEffectorPlatform:
            ArmLinkPointIsReadOnly = 0
            Arm1LinkPoint:
              Radius = 50
              Z = 0.0
            Arm2LinkPoint:
              Radius = 50
              Z = 0.0
            Arm3LinkPoint:
              Radius = 50
              Z = 0.0
            TranslationToFlangeIsReadOnly = 1
            TranslationToFlange:
              X = 0.0
              Y = 0.0
              Z = -44.5
        Offsets:
          JointAxisIsReadOnly = 1
          JointAxis[1] = 0.0
          JointAxis[2] = 0.0
          JointAxis[3] = 0.0
          JointAxis[4] = 0.0
        CountDirections:
          JointAxisIsReadOnly = 1
          JointAxis[1] = Standard
          JointAxis[2] = Standard
          JointAxis[3] = Standard
          JointAxis[4] = Standard
      CoordinatesNames = Default
        XCoordinateName = X
        YCoordinateName = Y
        ZCoordinateName = Z
        CCoordinateName = C
      WireFrameModelIsReadOnly = 0
      WireFrameModel = Standard
        UpperArm1IsReadOnly = 0
        UpperArm1 = ConnectionLine
          DistanceMin = -1.79769313486231E308
          DistanceMax = 1.79769313486231E308
          Distance = 5
        LowerArm1IsReadOnly = 0
        LowerArm1 = ConnectionLine
          DistanceMin = -1.79769313486231E308
          DistanceMax = 1.79769313486231E308
          Distance = 5
        UpperArm2IsReadOnly = 0
        UpperArm2 = ConnectionLine
          DistanceMin = -1.79769313486231E308
          DistanceMax = 1.79769313486231E308
          Distance = 5
        LowerArm2IsReadOnly = 0
        LowerArm2 = ConnectionLine
          DistanceMin = -1.79769313486231E308
          DistanceMax = 1.79769313486231E308
          Distance = 5
        UpperArm3IsReadOnly = 0
        UpperArm3 = ConnectionLine
          DistanceMin = -1.79769313486231E308
          DistanceMax = 1.79769313486231E308
          Distance = 5
        LowerArm3IsReadOnly = 0
        LowerArm3 = ConnectionLine
          DistanceMin = -1.79769313486231E308
          DistanceMax = 1.79769313486231E308
          Distance = 5
        EndEffectorPlatformToFlangeIsReadOnly = 0
        EndEffectorPlatformToFlange = ConnectionLine
          DistanceMin = -1.79769313486231E308
          DistanceMax = 1.79769313486231E308
          Distance = 5
        FlangeToTcp = NotUsed
      DynamicModelIsReadOnly = 0
      DynamicModel = DynParTable
        TableRef
      InternalDynamicModelIsReadOnly = 1
      InternalDynamicModel = Used
        TypeIsReadOnly = 1
        Type = D4-1100-S026-R100
        Row[1]:
          Index = 0
          Value = 4
          Unit = 
          Description = type of robot dyn par model
        Row[2]:
          Index = 1
          Value = 1.017
          Unit = kg
          Description = m1
        Row[3]:
          Index = 2
          Value = 0.10420182
          Unit = kgm
          Description = m1*rc1x
        Row[4]:
          Index = 3
          Value = 0
          Unit = kgm
          Description = m1*rc1y
        Row[5]:
          Index = 4
          Value = 0.00444429
          Unit = kgm
          Description = m1*rc1z
        Row[6]:
          Index = 5
          Value = 0
          Unit = kgm^2
          Description = m1*rc1x*rc1y
        Row[7]:
          Index = 6
          Value = 0
          Unit = kgm^2
          Description = m1*rc1y*rc1z
        Row[8]:
          Index = 7
          Value = 0.0004553619534
          Unit = kgm^2
          Description = m1*rc1x*rc1z
        Row[9]:
          Index = 8
          Value = 0.0106765184772
          Unit = kgm^2
          Description = m1*rc1x^2
        Row[10]:
          Index = 9
          Value = 0
          Unit = kgm^2
          Description = m1*rc1y^2
        Row[11]:
          Index = 10
          Value = 0.0000194215473
          Unit = kgm^2
          Description = m1*rc1z^2
        Row[12]:
          Index = 11
          Value = 0
          Unit = kgm^2
          Description = Jxx1
        Row[13]:
          Index = 12
          Value = 0.012935562
          Unit = kgm^2
          Description = Jyy1
        Row[14]:
          Index = 13
          Value = 0
          Unit = kgm^2
          Description = Jzz1
        Row[15]:
          Index = 14
          Value = 1.017
          Unit = kg
          Description = m2
        Row[16]:
          Index = 15
          Value = 0.10420182
          Unit = kgm
          Description = m2*rc2x
        Row[17]:
          Index = 16
          Value = 0
          Unit = kgm
          Description = m2*rc2y
        Row[18]:
          Index = 17
          Value = 0.00444429
          Unit = kgm
          Description = m2*rc2z
        Row[19]:
          Index = 18
          Value = 0
          Unit = kgm^2
          Description = m2*rc2x*rc2y
        Row[20]:
          Index = 19
          Value = 0
          Unit = kgm^2
          Description = m2*rc2y*rc2z
        Row[21]:
          Index = 20
          Value = 0.0004553619534
          Unit = kgm^2
          Description = m2*rc2x*rc2z
        Row[22]:
          Index = 21
          Value = 0.0106765184772
          Unit = kgm^2
          Description = m2*rc2x^2
        Row[23]:
          Index = 22
          Value = 0
          Unit = kgm^2
          Description = m2*rc2y^2
        Row[24]:
          Index = 23
          Value = 0.0000194215473
          Unit = kgm^2
          Description = m2*rc2z^2
        Row[25]:
          Index = 24
          Value = 0
          Unit = kgm^2
          Description = Jxx2
        Row[26]:
          Index = 25
          Value = 0.012935562
          Unit = kgm^2
          Description = Jyy2
        Row[27]:
          Index = 26
          Value = 0
          Unit = kgm^2
          Description = Jzz2
        Row[28]:
          Index = 27
          Value = 1.017
          Unit = kg
          Description = m3
        Row[29]:
          Index = 28
          Value = 0.10420182
          Unit = kgm
          Description = m3*rc3x
        Row[30]:
          Index = 29
          Value = 0
          Unit = kgm
          Description = m3*rc3y
        Row[31]:
          Index = 30
          Value = 0.00444429
          Unit = kgm
          Description = m3*rc3z
        Row[32]:
          Index = 31
          Value = 0
          Unit = kgm^2
          Description = m3*rc3x*rc3y
        Row[33]:
          Index = 32
          Value = 0
          Unit = kgm^2
          Description = m3*rc3y*rc3z
        Row[34]:
          Index = 33
          Value = 0.0004553619534
          Unit = kgm^2
          Description = m3*rc3x*rc3z
        Row[35]:
          Index = 34
          Value = 0.0106765184772
          Unit = kgm^2
          Description = m3*rc3x^2
        Row[36]:
          Index = 35
          Value = 0
          Unit = kgm^2
          Description = m3*rc3y^2
        Row[37]:
          Index = 36
          Value = 0.0000194215473
          Unit = kgm^2
          Description = m3*rc3z^2
        Row[38]:
          Index = 37
          Value = 0
          Unit = kgm^2
          Description = Jxx3
        Row[39]:
          Index = 38
          Value = 0.012935562
          Unit = kgm^2
          Description = Jyy3
        Row[40]:
          Index = 39
          Value = 0
          Unit = kgm^2
          Description = Jzz3
        Row[41]:
          Index = 40
          Value = 0.363
          Unit = kg
          Description = m4
        Row[42]:
          Index = 41
          Value = 0
          Unit = kgm
          Description = m4*rc4x
        Row[43]:
          Index = 42
          Value = 0
          Unit = kgm
          Description = m4*rc4y
        Row[44]:
          Index = 43
          Value = 0.154275
          Unit = kgm
          Description = m4*rc4z
        Row[45]:
          Index = 44
          Value = 0
          Unit = kgm^2
          Description = m4*rc4x*rc4y
        Row[46]:
          Index = 45
          Value = 0
          Unit = kgm^2
          Description = m4*rc4y*rc4z
        Row[47]:
          Index = 46
          Value = 0
          Unit = kgm^2
          Description = m4*rc4x*rc4z
        Row[48]:
          Index = 47
          Value = 0
          Unit = kgm^2
          Description = m4*rc4x^2
        Row[49]:
          Index = 48
          Value = 0
          Unit = kgm^2
          Description = m4*rc4y^2
        Row[50]:
          Index = 49
          Value = 0.154275
          Unit = kgm^2
          Description = m4*rc4z^2
        Row[51]:
          Index = 50
          Value = 0.037962996
          Unit = kgm^2
          Description = Jxx4
        Row[52]:
          Index = 51
          Value = 0.037962996
          Unit = kgm^2
          Description = Jyy4
        Row[53]:
          Index = 52
          Value = 0
          Unit = kgm^2
          Description = Jzz4
        Row[54]:
          Index = 53
          Value = 0.363
          Unit = kg
          Description = m5
        Row[55]:
          Index = 54
          Value = 0
          Unit = kgm
          Description = m5*rc5x
        Row[56]:
          Index = 55
          Value = 0
          Unit = kgm
          Description = m5*rc5y
        Row[57]:
          Index = 56
          Value = 0.154275
          Unit = kgm
          Description = m5*rc5z
        Row[58]:
          Index = 57
          Value = 0
          Unit = kgm^2
          Description = m5*rc5x*rc5y
        Row[59]:
          Index = 58
          Value = 0
          Unit = kgm^2
          Description = m5*rc5y*rc5z
        Row[60]:
          Index = 59
          Value = 0
          Unit = kgm^2
          Description = m5*rc5x*rc5z
        Row[61]:
          Index = 60
          Value = 0
          Unit = kgm^2
          Description = m5*rc5x^2
        Row[62]:
          Index = 61
          Value = 0
          Unit = kgm^2
          Description = m5*rc5y^2
        Row[63]:
          Index = 62
          Value = 0.154275
          Unit = kgm^2
          Description = m5*rc5z^2
        Row[64]:
          Index = 63
          Value = 0.037962996
          Unit = kgm^2
          Description = Jxx5
        Row[65]:
          Index = 64
          Value = 0.037962996
          Unit = kgm^2
          Description = Jyy5
        Row[66]:
          Index = 65
          Value = 0
          Unit = kgm^2
          Description = Jzz5
        Row[67]:
          Index = 66
          Value = 0.363
          Unit = kg
          Description = m6
        Row[68]:
          Index = 67
          Value = 0
          Unit = kgm
          Description = m6*rc6x
        Row[69]:
          Index = 68
          Value = 0
          Unit = kgm
          Description = m6*rc6y
        Row[70]:
          Index = 69
          Value = 0.154275
          Unit = kgm
          Description = m6*rc6z
        Row[71]:
          Index = 70
          Value = 0
          Unit = kgm^2
          Description = m6*rc6x*rc6y
        Row[72]:
          Index = 71
          Value = 0
          Unit = kgm^2
          Description = m6*rc6y*rc6z
        Row[73]:
          Index = 72
          Value = 0
          Unit = kgm^2
          Description = m6*rc6x*rc6z
        Row[74]:
          Index = 73
          Value = 0
          Unit = kgm^2
          Description = m6*rc6x^2
        Row[75]:
          Index = 74
          Value = 0
          Unit = kgm^2
          Description = m6*rc6y^2
        Row[76]:
          Index = 75
          Value = 0.154275
          Unit = kgm^2
          Description = m6*rc6z^2
        Row[77]:
          Index = 76
          Value = 0.037962996
          Unit = kgm^2
          Description = Jxx6
        Row[78]:
          Index = 77
          Value = 0.037962996
          Unit = kgm^2
          Description = Jyy6
        Row[79]:
          Index = 78
          Value = 0
          Unit = kgm^2
          Description = Jzz6
        Row[80]:
          Index = 79
          Value = 0.47
          Unit = kg
          Description = m7
        Row[81]:
          Index = 80
          Value = 0
          Unit = kgm
          Description = m7*rc7x
        Row[82]:
          Index = 81
          Value = 0
          Unit = kgm
          Description = m7*rc7y
        Row[83]:
          Index = 82
          Value = 0.14805
          Unit = kgm
          Description = m7*rc7z
        Row[84]:
          Index = 83
          Value = 0
          Unit = kgm^2
          Description = m7*rc7x*rc7y
        Row[85]:
          Index = 84
          Value = 0
          Unit = kgm^2
          Description = m7*rc7y*rc7z
        Row[86]:
          Index = 85
          Value = 0
          Unit = kgm^2
          Description = m7*rc7x*rc7z
        Row[87]:
          Index = 86
          Value = 0
          Unit = kgm^2
          Description = m7*rc7x^2
        Row[88]:
          Index = 87
          Value = 0
          Unit = kgm^2
          Description = m7*rc7y^2
        Row[89]:
          Index = 88
          Value = 0.04663575
          Unit = kgm^2
          Description = m7*rc7z^2
        Row[90]:
          Index = 89
          Value = 0.02385687
          Unit = kgm^2
          Description = Jxx7
        Row[91]:
          Index = 90
          Value = 0.02385687
          Unit = kgm^2
          Description = Jyy7
        Row[92]:
          Index = 91
          Value = 0.000187166
          Unit = kgm^2
          Description = Jzz7
        Row[93]:
          Index = 92
          Value = 0.408
          Unit = kg
          Description = m8
        Row[94]:
          Index = 93
          Value = 0
          Unit = kgm
          Description = m8*rc8x
        Row[95]:
          Index = 94
          Value = 0
          Unit = kgm
          Description = m8*rc8y
        Row[96]:
          Index = 95
          Value = 0.10608
          Unit = kgm
          Description = m8*rc8z
        Row[97]:
          Index = 96
          Value = 0
          Unit = kgm^2
          Description = m8*rc8x*rc8y
        Row[98]:
          Index = 97
          Value = 0
          Unit = kgm^2
          Description = m8*rc8y*rc8z
        Row[99]:
          Index = 98
          Value = 0
          Unit = kgm^2
          Description = m8*rc8x*rc8z
        Row[100]:
          Index = 99
          Value = 0
          Unit = kgm^2
          Description = m8*rc8x^2
        Row[101]:
          Index = 100
          Value = 0
          Unit = kgm^2
          Description = m8*rc8y^2
        Row[102]:
          Index = 101
          Value = 0.0275808
          Unit = kgm^2
          Description = m8*rc8z^2
        Row[103]:
          Index = 102
          Value = 0.019126177
          Unit = kgm^2
          Description = Jxx8
        Row[104]:
          Index = 103
          Value = 0.019126177
          Unit = kgm^2
          Description = Jyy8
        Row[105]:
          Index = 104
          Value = 0.000075111
          Unit = kgm^2
          Description = Jzz8
        Row[106]:
          Index = 105
          Value = 0.44
          Unit = kg
          Description = m9
        Row[107]:
          Index = 106
          Value = 0
          Unit = kgm
          Description = m9*rc9x
        Row[108]:
          Index = 107
          Value = 0
          Unit = kgm
          Description = m9*rc9y
        Row[109]:
          Index = 108
          Value = 0
          Unit = kgm
          Description = m9*rc9z
        Row[110]:
          Index = 109
          Value = 0
          Unit = kgm^2
          Description = m9*rc9x*rc9y
        Row[111]:
          Index = 110
          Value = 0
          Unit = kgm^2
          Description = m9*rc9y*rc9z
        Row[112]:
          Index = 111
          Value = 0
          Unit = kgm^2
          Description = m9*rc9x*rc9z
        Row[113]:
          Index = 112
          Value = 0
          Unit = kgm^2
          Description = m9*rc9x^2
        Row[114]:
          Index = 113
          Value = 0
          Unit = kgm^2
          Description = m9*rc9y^2
        Row[115]:
          Index = 114
          Value = 0
          Unit = kgm^2
          Description = m9*rc9z^2
        Row[116]:
          Index = 115
          Value = 0
          Unit = kgm^2
          Description = Jxx9
        Row[117]:
          Index = 116
          Value = 0
          Unit = kgm^2
          Description = Jyy9
        Row[118]:
          Index = 117
          Value = 0
          Unit = kgm^2
          Description = Jzz9
        Row[119]:
          Index = 118
          Value = 0
          Unit = kg
          Description = m10
        Row[120]:
          Index = 119
          Value = 0
          Unit = kgm
          Description = m10*rc10x
        Row[121]:
          Index = 120
          Value = 0
          Unit = kgm
          Description = m10*rc10y
        Row[122]:
          Index = 121
          Value = 0
          Unit = kgm
          Description = m10*rc10z
        Row[123]:
          Index = 122
          Value = 0
          Unit = kgm^2
          Description = m10*rc10x*rc10y
        Row[124]:
          Index = 123
          Value = 0
          Unit = kgm^2
          Description = m10*rc10y*rc10z
        Row[125]:
          Index = 124
          Value = 0
          Unit = kgm^2
          Description = m10*rc10x*rc10z
        Row[126]:
          Index = 125
          Value = 0
          Unit = kgm^2
          Description = m10*rc10x^2
        Row[127]:
          Index = 126
          Value = 0
          Unit = kgm^2
          Description = m10*rc10y^2
        Row[128]:
          Index = 127
          Value = 0
          Unit = kgm^2
          Description = m10*rc10z^2
        Row[129]:
          Index = 128
          Value = 0
          Unit = kgm^2
          Description = Jxx10
        Row[130]:
          Index = 129
          Value = 0
          Unit = kgm^2
          Description = Jyy10
        Row[131]:
          Index = 130
          Value = 0.000044599
          Unit = kgm^2
          Description = Jzz10
        Row[132]:
          Index = 144
          Value = 0.000393
          Unit = kgm^2
          Description = JDrive1
        Row[133]:
          Index = 145
          Value = 0.000393
          Unit = kgm^2
          Description = JDrive2
        Row[134]:
          Index = 146
          Value = 0.000393
          Unit = kgm^2
          Description = JDrive3
        Row[135]:
          Index = 147
          Value = 0.000092
          Unit = kgm^2
          Description = JDrive4
        Row[136]:
          Index = 148
          Value = 0.249554950768092
          Unit = Nms
          Description = dV1
        Row[137]:
          Index = 149
          Value = 0.249554950768092
          Unit = Nms
          Description = dV2
        Row[138]:
          Index = 150
          Value = 0.249554950768092
          Unit = Nms
          Description = dV3
        Row[139]:
          Index = 151
          Value = 1.59154943091895E-02
          Unit = Nms
          Description = dV4
        Row[140]:
          Index = 152
          Value = 6.16
          Unit = Nm
          Description = dC1
        Row[141]:
          Index = 153
          Value = 6.16
          Unit = Nm
          Description = dC2
        Row[142]:
          Index = 154
          Value = 6.16
          Unit = Nm
          Description = dC3
        Row[143]:
          Index = 155
          Value = 1
          Unit = Nm
          Description = dC4
      DynamicLimits = DynParTables
        GearboxLimitsTableRef
        CrossSectionLimitsTableRef
      InternalDynamicLimits = Used
        TypeIsReadOnly = 1
        Type = D4-1100-S026-R100
        GearboxLimits:
          Row[1]:
            Index = 0
            Value = 4
            Unit = 
            Description = Type of robot dyn par model
          Row[2]:
            Index = 1
            Value = 85
            Unit = Nm
            Description = Gearbox Drive 1
          Row[3]:
            Index = 2
            Value = 85
            Unit = Nm
            Description = Gearbox Drive 2
          Row[4]:
            Index = 3
            Value = 85
            Unit = Nm
            Description = Gearbox Drive 3
          Row[5]:
            Index = 4
            Value = 3.5
            Unit = Nm
            Description = Gearbox Drive 4
        CrossSectionLimits:
          Row[1]:
            Index = 0
            Value = 4
            Unit = Variant
            Description = 
          Row[2]:
            Index = 1
            Value = 10000
            Unit = N
            Description = 
          Row[3]:
            Index = 2
            Value = 10000
            Unit = N
            Description = 
          Row[4]:
            Index = 3
            Value = 10000
            Unit = N
            Description = 
          Row[5]:
            Index = 4
            Value = 10000
            Unit = Nm
            Description = 
          Row[6]:
            Index = 5
            Value = 10000
            Unit = Nm
            Description = 
          Row[7]:
            Index = 6
            Value = 10000
            Unit = Nm
            Description = 
          Row[8]:
            Index = 7
            Value = 225
            Unit = N
            Description = 
          Row[9]:
            Index = 8
            Value = 225
            Unit = N
            Description = 
          Row[10]:
            Index = 9
            Value = 225
            Unit = N
            Description = 
          Row[11]:
            Index = 10
            Value = 225
            Unit = N
            Description = 
          Row[12]:
            Index = 11
            Value = 225
            Unit = N
            Description = 
          Row[13]:
            Index = 12
            Value = 225
            Unit = N
            Description = 
      LoadDependentJerkLimitsIsReadOnly = 1
      LoadDependentJerkLimits = PayloadDependentJerkReduction
        JerkReduction[1]:
          PayloadInKgIsReadOnly = 0
          PayloadInKg = 0
          JerkReductionInPercentIsReadOnly = 0
          JerkReductionInPercent = 0
        JerkReduction[2]:
          PayloadInKgIsReadOnly = 0
          PayloadInKg = 0.35
          JerkReductionInPercentIsReadOnly = 0
          JerkReductionInPercent = 0
        JerkReduction[3]:
          PayloadInKgIsReadOnly = 0
          PayloadInKg = 1
          JerkReductionInPercentIsReadOnly = 0
          JerkReductionInPercent = 50
        JerkReduction[4]:
          PayloadInKgIsReadOnly = 0
          PayloadInKg = 1.5
          JerkReductionInPercentIsReadOnly = 0
          JerkReductionInPercent = 50
        JerkReduction[5]:
          PayloadInKgIsReadOnly = 0
          PayloadInKg = 3
          JerkReductionInPercentIsReadOnly = 0
          JerkReductionInPercent = 70
      CouplingsIsInvisible = 0
      JointAxesPositionLimits:
        JointAxisIsReadOnly = 1
        JointAxis[1] = UseAxisLimits
        JointAxis[2] = UseAxisLimits
        JointAxis[3] = UseAxisLimits
        JointAxis[4] = UseAxisLimits
      WorkingRangeIsReadOnly = 1
      WorkingRange = Standard
        ScnObjWorkRangeCfg = Visible
          Top:
            LineWidth = 0.25
            Opacitiy = 0.25
            LineColor:
              Red = 0.0
              Green = 0.75
              Blue = 0.0
            Style = 2
            JoinToParent = TRUE
          MidSegment:
            LineWidth = 0.25
            Opacitiy = 0.25
            LineColor:
              Red = 0.0
              Green = 0.75
              Blue = 0.0
            Style = 2
            JoinToParent = TRUE
          BottomSegment:
            LineWidth = 0.25
            Opacitiy = 0.25
            LineColor:
              Red = 0.0
              Green = 0.75
              Blue = 0.0
            Style = 2
            JoinToParent = TRUE
        BaseToTopIsReadOnly = 1
        BaseToTop = 706.0
        TopHeightIsReadOnly = 1
        MiddleHeightIsReadOnly = 1
        MiddleHeight = 250.0
        BottomHeightIsReadOnly = 1
        BottomHeight = 150.0
        TopRadiusIsReadOnly = 1
        TopRadius = 550.0
        MiddleRadiusIsReadOnly = 1
        MiddleRadius = 550.0
        BottomRadiusIsReadOnly = 1
        BottomRadius = 335.75
```

### Config_5.axesgroupfeature - 5APC3100_KBU3_000/mappMotion/Codian_D4r1100R_1/Config_5.axesgroupfeature
```
Element Feature_Programs_D4r1100R_1 (Type=axesgroupfeature)
  Type = Program
    ModalDataBehaviour = UseAxesGroupSettings
    InitialSettings:
      InterpolationTypes = LinearRapid
      PositionCoordinates = Absolute
      CircleCoordinates = Relative
      JACS_ACSProgramming = JACS
      ContourConnection = Inactive
      AccuracyHoldDelays = None
      ProgrammingUnits = UseAxesGroupSettings
      Feedrates:
        FeedPath = Standard
        FeedCharacteristic = StandardCharacteristic
        FeedType = Feedrate
        FeedReduction = Inactive
        FeedrateValue = 0.0
        InverseFeedrateValue = 0.0
        FeedratePerRevValue = 0.0
    DefaultLanguage = BRGCode
    Location = User
      UserLocation[1]:
        FileDevice = GProgram_SIM
      UserLocation[2]:
        FileDevice = GProgram
    ProgramElements:
      PVs:
        PV[1]:
          PvName = ::APP_Robot1:BeltSpeed
          Advanced:
            Alias = BeltSpeed
            Synchronization = Ip
            Reference = No
        PV[2]:
          PvName = ::APP_Robot1:XRobotPos
          Advanced:
            Alias = XRobotPos
            Synchronization = Ip
            Reference = No
        PV[3]:
          PvName = ::APP_Robot1:YRobotPos
          Advanced:
            Alias = YRobotPos
            Synchronization = Ip
            Reference = No
        PV[4]:
          PvName = ::APP_Robot1:XRobotOfs
          Advanced:
            Alias = XRobotOfs
            Synchronization = Ip
            Reference = No
        PV[5]:
          PvName = ::APP_Robot1:MaxPickPosX
          Advanced:
            Alias = MaxPickPosX
            Synchronization = Ip
            Reference = No
        PV[6]:
          PvName = ::APP_Robot1:NextTrackingObject
          Advanced:
            Alias = NextTrackingObject
            Synchronization = Ip
            Reference = No
        PV[7]:
          PvName = ::APP_Robot1:MinPickPosX
          Advanced:
            Alias = MinPickPosX
            Synchronization = Ip
            Reference = No
        PV[8]:
          PvName = ::APP_Robot1:MinWorkspaceX
          Advanced:
            Alias = MinWorkspaceX
            Synchronization = Ip
            Reference = No
```

### Config_8.axesgroup - 5APC3100_KBU3_000/mappMotion/Codian_D4r1100R_1/Config_8.axesgroup
```
Element gAxesGroup_D4r1100R_1 (Type=axesgroup)
  Type = PathGenAxesGroup
    ProcessingTaskClass = 1
    PhysicalAxes:
      JointAxes:
        JointAxis[1]:
          AxisRef = gAxisQ1_D4r1100R_1
        JointAxis[2]:
          AxisRef = gAxisQ2_D4r1100R_1
        JointAxis[3]:
          AxisRef = gAxisQ3_D4r1100R_1
        JointAxis[4]:
          Name = QC
          AxisRef = gAxisQC_D4r1100R_1
    MechanicalSystem:
      MechSysRef = MechSys_D4r1100R_1
    BasicSettings:
      GeometryPlanning:
        MaxTangentialTransitionDeviation = 0.05
      TrajectoryPlanning:
        LimitCheckResolution:
          Time = 0.005
        BufferTime:
          Time = 0.05
      Miscellaneous:
        TimeStretchOverride:
          JerkSuppression = Basic
            AdaptationTime = 0.3
    StopReaction:
      AxisError:
        AxisReaction = DynamicStop
    AxesGroupFeatures:
      FeatureRef[1] = Feature_Programs
      FeatureRef[2] = Feature_FrameHierachy
      FeatureRef[3] = Feature_MFunctions
      FeatureRef[4] = Feature_PathDefRobot
      FeatureRef[5] = Feature_Selection
      FeatureRef[6] = Feature_TrackingRobot
      FeatureRef[7] = Feature_WorkspaceMonitoring
```

### Config_2.axesgroup - 5APC3100_KBU3_000/mappMotion/Codian_D4r1100_1/Config_2.axesgroup
```
Element gAxesGroup_D4r1100_1 (Type=axesgroup)
  Type = PathGenAxesGroup
    ProcessingTaskClass = 1
    License = 1
    PhysicalAxes:
      JointAxes:
        JointAxisAxisRefIsReadOnly = 0
        JointAxis[1]:
          Name = Q1
          AxisRef = gAxisQ1_D4r1100_1
        JointAxis[2]:
          Name = Q2
          AxisRef = gAxisQ2_D4r1100_1
        JointAxis[3]:
          Name = Q3
          AxisRef = gAxisQ3_D4r1100_1
    MechanicalSystem:
      MechSysRefIsReadOnly = 0
      MechSysRef = MechSys_D4r1100_1
    BasicSettings:
      ModalDataBehaviour = ResetToDefault
      GeometryPlanning:
        TCPResolutionIsReadOnly = 0
        TCPResolution:
          LengthResolution = 0.001
          AngleResolution = 0.001
        Rounding:
          PathDistance = 0.0
          SymmetricRounding = Yes
          LastSegment = Half
          AvoidZeroCurvature = No
        RoundingMode = Standard
        MaxCornerDeviation = 0.0
        MaxTangentialTransitionDeviation = 0.05
        MaxRadiusDeviation = 0.001
        WorkingPlane = XY
      TrajectoryPlanningIsReadOnly = 0
      TrajectoryPlanning = Basic
        LimitCheckResolutionIsReadOnly = 0
        LimitCheckResolution = UserDefinedTime
          TimeIsReadOnly = 0
          Time = 0.005
        BufferTime = UserDefinedTime
          Time = 0.05
        BarrierParametrization = JointCoordinates
        TorqueLimitConsideration = Exact
      Miscellaneous:
        NonMovementsLimit = NotUsed
        TimeStretchOverride:
          JerkSuppression = NotUsed
    StopReaction:
      AxisError:
        AxisReactionIsReadOnly = 0
    AxesGroupFeatures:
      FeatureRef[1] = Feature_Programs_D4r1100_1
      FeatureRef[2] = Feature_FrameHierachy
      FeatureRef[3] = Feature_InterpreterLog
      FeatureRef[4] = Feature_MFunctions
      FeatureRef[5] = Feature_Monitoring
      FeatureRef[6] = Feature_PathDefRobot
      FeatureRef[7] = Feature_TrackingRobot
      FeatureRef[8] = Feature_WorkspaceMonitoring
    SceneObject:
      FileDevice = ComponentScenes
      FileNamePrefix = PathGen_
      FrameSize = 150
      FrameName = Invisible
      Positioner = NotUsed
      Object = Visible
      Boundaries = NotUsed
  Alarms = None
```

### Config_3.axis - 5APC3100_KBU3_000/mappMotion/Codian_D4r1100_1/Config_3.axis
```
Element gAxisQ1_D4r1100_1 (Type=axis)
  BaseTypeIsReadOnly = 0
  BaseType = RotaryBounded
    MeasurementUnitIsReadOnly = 1
    MeasurementUnit = 17476
    MeasurementResolutionIsReadOnly = 1
    MeasurementResolution = 0.001
    CountDirectionIsReadOnly = 1
    CountDirection = Inverse
  MovementLimitsIsReadOnly = 0
  MovementLimits = InternalForPathControlledAxis
    Position:
      LowerLimitMin = -47
      UpperLimitMax = 100
      LowerLimit = -47
      UpperLimit = 100
    VelocityIsReadOnly = 0
    Velocity:
      VelocityMax = 3.4E38
      Velocity = 1160
    AccelerationIsReadOnly = 0
    Acceleration:
      AccelerationMax = 3.4E38
      Acceleration = 11600
    DecelerationIsReadOnly = 0
    Deceleration:
      DecelerationMax = 3.4E38
      Deceleration = 11600
    JerkIsReadOnly = 0
    Jerk = Advanced
      JerkAccelerationPositiveMin = 0
      JerkAccelerationPositiveMax = 3.4E38
      JerkAccelerationPositive = 2200000
      JerkAccelerationNegativeMin = 0
      JerkAccelerationNegativeMax = 3.4E38
      JerkAccelerationNegative = 2200000
      JerkDecelerationPositiveMin = 0
      JerkDecelerationPositiveMax = 3.4E38
      JerkDecelerationPositive = 2000000
      JerkDecelerationNegativeMin = 0
      JerkDecelerationNegativeMax = 3.4E38
      JerkDecelerationNegative = 2000000
    TorqueIsInvisible = 0
    TorqueIsReadOnly = 0
    Torque = Basic
      TorqueMax = 3.4E38
      Torque = 20.5
  Alarms = None
Element gAxisQ2_D4r1100_1 (Type=axis)
  BaseTypeIsReadOnly = 0
  BaseType = RotaryBounded
    MeasurementUnitIsReadOnly = 1
    MeasurementUnit = 17476
    MeasurementResolutionIsReadOnly = 1
    MeasurementResolution = 0.001
    CountDirectionIsReadOnly = 1
    CountDirection = Inverse
  MovementLimitsIsReadOnly = 0
  MovementLimits = InternalForPathControlledAxis
    Position:
      LowerLimitMin = -47
      UpperLimitMax = 100
      LowerLimit = -47
      UpperLimit = 100
    VelocityIsReadOnly = 0
    Velocity:
      VelocityMax = 3.4E38
      Velocity = 1160
    AccelerationIsReadOnly = 0
    Acceleration:
      AccelerationMax = 3.4E38
      Acceleration = 11600
    DecelerationIsReadOnly = 0
    Deceleration:
      DecelerationMax = 3.4E38
      Deceleration = 35000
    JerkIsReadOnly = 0
    Jerk = Advanced
      JerkAccelerationPositiveMin = 0
      JerkAccelerationPositiveMax = 3.4E38
      JerkAccelerationPositive = 2200000
      JerkAccelerationNegativeMin = 0
      JerkAccelerationNegativeMax = 3.4E38
      JerkAccelerationNegative = 2200000
      JerkDecelerationPositiveMin = 0
      JerkDecelerationPositiveMax = 3.4E38
      JerkDecelerationPositive = 2000000
      JerkDecelerationNegativeMin = 0
      JerkDecelerationNegativeMax = 3.4E38
      JerkDecelerationNegative = 2000000
    TorqueIsInvisible = 0
    TorqueIsReadOnly = 0
    Torque = Basic
      TorqueMax = 3.4E38
      Torque = 20.5
  Alarms = None
Element gAxisQ3_D4r1100_1 (Type=axis)
  BaseTypeIsReadOnly = 0
  BaseType = RotaryBounded
    MeasurementUnitIsReadOnly = 1
    MeasurementUnit = 17476
    MeasurementResolutionIsReadOnly = 1
    MeasurementResolution = 0.001
    CountDirectionIsReadOnly = 1
    CountDirection = Inverse
  MovementLimitsIsReadOnly = 0
  MovementLimits = InternalForPathControlledAxis
    Position:
      LowerLimitMin = -47
      UpperLimitMax = 100
      LowerLimit = -47
      UpperLimit = 100
    VelocityIsReadOnly = 0
    Velocity:
      VelocityMax = 3.4E38
      Velocity = 1160
    AccelerationIsReadOnly = 0
    Acceleration:
      AccelerationMax = 3.4E38
      Acceleration = 11600
    DecelerationIsReadOnly = 0
    Deceleration:
      DecelerationMax = 3.4E38
      Deceleration = 11600
    JerkIsReadOnly = 0
    Jerk = Advanced
      JerkAccelerationPositiveMin = 0
      JerkAccelerationPositiveMax = 3.4E38
      JerkAccelerationPositive = 2200000
      JerkAccelerationNegativeMin = 0
      JerkAccelerationNegativeMax = 3.4E38
      JerkAccelerationNegative = 2200000
      JerkDecelerationPositiveMin = 0
      JerkDecelerationPositiveMax = 3.4E38
      JerkDecelerationPositive = 2000000
      JerkDecelerationNegativeMin = 0
      JerkDecelerationNegativeMax = 3.4E38
      JerkDecelerationNegative = 2000000
    TorqueIsInvisible = 0
    TorqueIsReadOnly = 0
    Torque = Basic
      TorqueMax = 3.4E38
      Torque = 20.5
  Alarms = None
```

### Config_4.mechanicalsystem - 5APC3100_KBU3_000/mappMotion/Codian_D4r1100_1/Config_4.mechanicalsystem
```
Element MechSys_D4r1100_1 (Type=mechanicalsystem)
  TypeIsReadOnly = 1
  Type = Delta
    SubtypeIsReadOnly = 1
    Subtype = 3AxesDeltaA
      SceneViewerObject = ObjectID
        ID = 1390
      DescriptionIsReadOnly = 1
      Description = Standard
        Dimensions:
          BasePlatform:
            CenterIsReadOnly = 0
            Center:
              X = 0.0
              Y = 0.0
              Z = 0
            ArmLinkPointIsReadOnly = 0
            Arm1LinkPoint:
              Angle = 0.0
              Radius = 200
              Z = -90
            Arm2LinkPoint:
              Angle = -120.0
              Radius = 200
              Z = -90
            Arm3LinkPoint:
              Angle = -240.0
              Radius = 200
              Z = -90
          Arms:
            ArmIsReadOnly = 0
            Arm1:
              UpperArmLength = 320
              LowerArmLength = 850
            Arm2:
              UpperArmLength = 320
              LowerArmLength = 850
            Arm3:
              UpperArmLength = 320
              LowerArmLength = 850
            LowerArmPairDistance = 125
          EndEffectorPlatform:
            ArmLinkPointIsReadOnly = 0
            Arm1LinkPoint:
              Radius = 50
              Z = 0.0
            Arm2LinkPoint:
              Radius = 50
              Z = 0.0
            Arm3LinkPoint:
              Radius = 50
              Z = 0.0
            TranslationToFlangeIsReadOnly = 1
            TranslationToFlange:
              X = 0.0
              Y = 0.0
              Z = -44.5
        Offsets:
          JointAxisIsReadOnly = 0
          JointAxis[1] = 0.0
          JointAxis[2] = 0.0
          JointAxis[3] = 0.0
        CountDirections:
          JointAxisIsReadOnly = 0
          JointAxis[1] = Standard
          JointAxis[2] = Standard
          JointAxis[3] = Standard
      CoordinatesNames = Default
        XCoordinateName = X
        YCoordinateName = Y
        ZCoordinateName = Z
      WireFrameModelIsReadOnly = 0
      WireFrameModel = Standard
        UpperArm1IsReadOnly = 0
        UpperArm1 = ConnectionLine
          DistanceMin = -1.79769313486231E308
          DistanceMax = 1.79769313486231E308
          Distance = 5
        LowerArm1IsReadOnly = 0
        LowerArm1 = ConnectionLine
          DistanceMin = -1.79769313486231E308
          DistanceMax = 1.79769313486231E308
          Distance = 5
        UpperArm2IsReadOnly = 0
        UpperArm2 = ConnectionLine
          DistanceMin = -1.79769313486231E308
          DistanceMax = 1.79769313486231E308
          Distance = 5
        LowerArm2IsReadOnly = 0
        LowerArm2 = ConnectionLine
          DistanceMin = -1.79769313486231E308
          DistanceMax = 1.79769313486231E308
          Distance = 5
        UpperArm3IsReadOnly = 0
        UpperArm3 = ConnectionLine
          DistanceMin = -1.79769313486231E308
          DistanceMax = 1.79769313486231E308
          Distance = 5
        LowerArm3IsReadOnly = 0
        LowerArm3 = ConnectionLine
          DistanceMin = -1.79769313486231E308
          DistanceMax = 1.79769313486231E308
          Distance = 5
        EndEffectorPlatformToFlangeIsReadOnly = 0
        EndEffectorPlatformToFlange = ConnectionLine
          DistanceMin = -1.79769313486231E308
          DistanceMax = 1.79769313486231E308
          Distance = 5
        FlangeToTcp = NotUsed
      DynamicModelIsReadOnly = 0
      DynamicModel = DynParTable
        TableRef
      InternalDynamicModelIsReadOnly = 1
      InternalDynamicModel = Used
        TypeIsReadOnly = 1
        Type = D4-1100-S026
        Row[1]:
          Index = 0
          Value = 3
          Unit = 
          Description = type of robot dyn par model
        Row[2]:
          Index = 1
          Value = 1.017
          Unit = kg
          Description = m1
        Row[3]:
          Index = 2
          Value = 0.10420182
          Unit = kgm
          Description = m1*rc1x
        Row[4]:
          Index = 3
          Value = 0
          Unit = kgm
          Description = m1*rc1y
        Row[5]:
          Index = 4
          Value = 0.00444429
          Unit = kgm
          Description = m1*rc1z
        Row[6]:
          Index = 5
          Value = 0
          Unit = kgm^2
          Description = m1*rc1x*rc1y
        Row[7]:
          Index = 6
          Value = 0
          Unit = kgm^2
          Description = m1*rc1y*rc1z
        Row[8]:
          Index = 7
          Value = 0.0004553619534
          Unit = kgm^2
          Description = m1*rc1x*rc1z
        Row[9]:
          Index = 8
          Value = 0.0106765184772
          Unit = kgm^2
          Description = m1*rc1x^2
        Row[10]:
          Index = 9
          Value = 0
          Unit = kgm^2
          Description = m1*rc1y^2
        Row[11]:
          Index = 10
          Value = 0.0000194215473
          Unit = kgm^2
          Description = m1*rc1z^2
        Row[12]:
          Index = 11
          Value = 0
          Unit = kgm^2
          Description = Jxx1
        Row[13]:
          Index = 12
          Value = 0.0129
          Unit = kgm^2
          Description = Jyy1
        Row[14]:
          Index = 13
          Value = 0
          Unit = kgm^2
          Description = Jzz1
        Row[15]:
          Index = 14
          Value = 1.017
          Unit = kg
          Description = m2
        Row[16]:
          Index = 15
          Value = 0.10420182
          Unit = kgm
          Description = m2*rc2x
        Row[17]:
          Index = 16
          Value = 0
          Unit = kgm
          Description = m2*rc2y
        Row[18]:
          Index = 17
          Value = 0.00444429
          Unit = kgm
          Description = m2*rc2z
        Row[19]:
          Index = 18
          Value = 0
          Unit = kgm^2
          Description = m2*rc2x*rc2y
        Row[20]:
          Index = 19
          Value = 0
          Unit = kgm^2
          Description = m2*rc2y*rc2z
        Row[21]:
          Index = 20
          Value = 0.0004553619534
          Unit = kgm^2
          Description = m2*rc2x*rc2z
        Row[22]:
          Index = 21
          Value = 0.0106765184772
          Unit = kgm^2
          Description = m2*rc2x^2
        Row[23]:
          Index = 22
          Value = 0
          Unit = kgm^2
          Description = m2*rc2y^2
        Row[24]:
          Index = 23
          Value = 0.0000194215473
          Unit = kgm^2
          Description = m2*rc2z^2
        Row[25]:
          Index = 24
          Value = 0
          Unit = kgm^2
          Description = Jxx2
        Row[26]:
          Index = 25
          Value = 0.0129
          Unit = kgm^2
          Description = Jyy2
        Row[27]:
          Index = 26
          Value = 0
          Unit = kgm^2
          Description = Jzz2
        Row[28]:
          Index = 27
          Value = 1.017
          Unit = kg
          Description = m3
        Row[29]:
          Index = 28
          Value = 0
          Unit = kgm
          Description = m3*rc3x
        Row[30]:
          Index = 29
          Value = 0
          Unit = kgm
          Description = m3*rc3y
        Row[31]:
          Index = 30
          Value = 0
          Unit = kgm
          Description = m3*rc3z
        Row[32]:
          Index = 31
          Value = 0
          Unit = kgm^2
          Description = m3*rc3x*rc3y
        Row[33]:
          Index = 32
          Value = 0
          Unit = kgm^2
          Description = m3*rc3y*rc3z
        Row[34]:
          Index = 33
          Value = 0
          Unit = kgm^2
          Description = m3*rc3x*rc3z
        Row[35]:
          Index = 34
          Value = 0
          Unit = kgm^2
          Description = m3*rc3x^2
        Row[36]:
          Index = 35
          Value = 0
          Unit = kgm^2
          Description = m3*rc3y^2
        Row[37]:
          Index = 36
          Value = 0
          Unit = kgm^2
          Description = m3*rc3z^2
        Row[38]:
          Index = 37
          Value = 0
          Unit = kgm^2
          Description = Jxx3
        Row[39]:
          Index = 38
          Value = 0.0129
          Unit = kgm^2
          Description = Jyy3
        Row[40]:
          Index = 39
          Value = 0
          Unit = kgm^2
          Description = Jzz3
        Row[41]:
          Index = 40
          Value = 0.363
          Unit = kg
          Description = m4
        Row[42]:
          Index = 41
          Value = 0
          Unit = kgm
          Description = m4*rc4x
        Row[43]:
          Index = 42
          Value = 0
          Unit = kgm
          Description = m4*rc4y
        Row[44]:
          Index = 43
          Value = 0
          Unit = kgm
          Description = m4*rc4z
        Row[45]:
          Index = 44
          Value = 0
          Unit = kgm^2
          Description = m4*rc4x*rc4y
        Row[46]:
          Index = 45
          Value = 0
          Unit = kgm^2
          Description = m4*rc4y*rc4z
        Row[47]:
          Index = 46
          Value = 0
          Unit = kgm^2
          Description = m4*rc4x*rc4z
        Row[48]:
          Index = 47
          Value = 0
          Unit = kgm^2
          Description = m4*rc4x^2
        Row[49]:
          Index = 48
          Value = 0
          Unit = kgm^2
          Description = m4*rc4y^2
        Row[50]:
          Index = 49
          Value = 0
          Unit = kgm^2
          Description = m4*rc4z^2
        Row[51]:
          Index = 50
          Value = 0.038
          Unit = kgm^2
          Description = Jxx4
        Row[52]:
          Index = 51
          Value = 0.038
          Unit = kgm^2
          Description = Jyy4
        Row[53]:
          Index = 52
          Value = 0
          Unit = kgm^2
          Description = Jzz4
        Row[54]:
          Index = 53
          Value = 0.363
          Unit = kg
          Description = m5
        Row[55]:
          Index = 54
          Value = 0
          Unit = kgm
          Description = m5*rc5x
        Row[56]:
          Index = 55
          Value = 0
          Unit = kgm
          Description = m5*rc5y
        Row[57]:
          Index = 56
          Value = 0
          Unit = kgm
          Description = m5*rc5z
        Row[58]:
          Index = 57
          Value = 0
          Unit = kgm^2
          Description = m5*rc5x*rc5y
        Row[59]:
          Index = 58
          Value = 0
          Unit = kgm^2
          Description = m5*rc5y*rc5z
        Row[60]:
          Index = 59
          Value = 0
          Unit = kgm^2
          Description = m5*rc5x*rc5z
        Row[61]:
          Index = 60
          Value = 0
          Unit = kgm^2
          Description = m5*rc5x^2
        Row[62]:
          Index = 61
          Value = 0
          Unit = kgm^2
          Description = m5*rc5y^2
        Row[63]:
          Index = 62
          Value = 0
          Unit = kgm^2
          Description = m5*rc5z^2
        Row[64]:
          Index = 63
          Value = 0.038
          Unit = kgm^2
          Description = Jxx5
        Row[65]:
          Index = 64
          Value = 0.038
          Unit = kgm^2
          Description = Jyy5
        Row[66]:
          Index = 65
          Value = 0
          Unit = kgm^2
          Description = Jzz5
        Row[67]:
          Index = 66
          Value = 0.363
          Unit = kg
          Description = m6
        Row[68]:
          Index = 67
          Value = 0
          Unit = kgm
          Description = m6*rc6x
        Row[69]:
          Index = 68
          Value = 0
          Unit = kgm
          Description = m6*rc6y
        Row[70]:
          Index = 69
          Value = 0
          Unit = kgm
          Description = m6*rc6z
        Row[71]:
          Index = 70
          Value = 0
          Unit = kgm^2
          Description = m6*rc6x*rc6y
        Row[72]:
          Index = 71
          Value = 0
          Unit = kgm^2
          Description = m6*rc6y*rc6z
        Row[73]:
          Index = 72
          Value = 0
          Unit = kgm^2
          Description = m6*rc6x*rc6z
        Row[74]:
          Index = 73
          Value = 0
          Unit = kgm^2
          Description = m6*rc6x^2
        Row[75]:
          Index = 74
          Value = 0
          Unit = kgm^2
          Description = m6*rc6y^2
        Row[76]:
          Index = 75
          Value = 0
          Unit = kgm^2
          Description = m6*rc6z^2
        Row[77]:
          Index = 76
          Value = 0.038
          Unit = kgm^2
          Description = Jxx6
        Row[78]:
          Index = 77
          Value = 0.038
          Unit = kgm^2
          Description = Jyy6
        Row[79]:
          Index = 78
          Value = 0
          Unit = kgm^2
          Description = Jzz6
        Row[80]:
          Index = 79
          Value = 0.374
          Unit = kg
          Description = m7
        Row[81]:
          Index = 80
          Value = 0
          Unit = kgm
          Description = m7*rc7x
        Row[82]:
          Index = 81
          Value = 0
          Unit = kgm
          Description = m7*rc7y
        Row[83]:
          Index = 82
          Value = 0
          Unit = kgm
          Description = m7*rc7z
        Row[84]:
          Index = 83
          Value = 0
          Unit = kgm^2
          Description = m7*rc7x*rc7y
        Row[85]:
          Index = 84
          Value = 0
          Unit = kgm^2
          Description = m7*rc7y*rc7z
        Row[86]:
          Index = 85
          Value = 0
          Unit = kgm^2
          Description = m7*rc7x*rc7z
        Row[87]:
          Index = 86
          Value = 0
          Unit = kgm^2
          Description = m7*rc7x^2
        Row[88]:
          Index = 87
          Value = 0
          Unit = kgm^2
          Description = m7*rc7y^2
        Row[89]:
          Index = 88
          Value = 0
          Unit = kgm^2
          Description = m7*rc7z^2
        Row[90]:
          Index = 89
          Value = 0
          Unit = kgm^2
          Description = Jxx7
        Row[91]:
          Index = 90
          Value = 0
          Unit = kgm^2
          Description = Jyy7
        Row[92]:
          Index = 91
          Value = 0
          Unit = kgm^2
          Description = Jzz7
        Row[93]:
          Index = 92
          Value = 0
          Unit = kg
          Description = m8
        Row[94]:
          Index = 93
          Value = 0
          Unit = kgm
          Description = m8*rc8x
        Row[95]:
          Index = 94
          Value = 0
          Unit = kgm
          Description = m8*rc8y
        Row[96]:
          Index = 95
          Value = 0
          Unit = kgm
          Description = m8*rc8z
        Row[97]:
          Index = 96
          Value = 0
          Unit = kgm^2
          Description = m8*rc8x*rc8y
        Row[98]:
          Index = 97
          Value = 0
          Unit = kgm^2
          Description = m8*rc8y*rc8z
        Row[99]:
          Index = 98
          Value = 0
          Unit = kgm^2
          Description = m8*rc8x*rc8z
        Row[100]:
          Index = 99
          Value = 0
          Unit = kgm^2
          Description = m8*rc8x^2
        Row[101]:
          Index = 100
          Value = 0
          Unit = kgm^2
          Description = m8*rc8y^2
        Row[102]:
          Index = 101
          Value = 0
          Unit = kgm^2
          Description = m8*rc8z^2
        Row[103]:
          Index = 102
          Value = 0
          Unit = kgm^2
          Description = Jxx8
        Row[104]:
          Index = 103
          Value = 0
          Unit = kgm^2
          Description = Jyy8
        Row[105]:
          Index = 104
          Value = 0
          Unit = kgm^2
          Description = Jzz8
        Row[106]:
          Index = 118
          Value = 0.000393
          Unit = kgm^2
          Description = JDrive1
        Row[107]:
          Index = 119
          Value = 0.000393
          Unit = kgm^2
          Description = JDrive2
        Row[108]:
          Index = 120
          Value = 0.000393
          Unit = kgm^2
          Description = JDrive3
        Row[109]:
          Index = 121
          Value = 0.249554950768092
          Unit = Nms
          Description = dV1
        Row[110]:
          Index = 122
          Value = 0.249554950768092
          Unit = Nms
          Description = dV2
        Row[111]:
          Index = 123
          Value = 0.249554950768092
          Unit = Nms
          Description = dV3
        Row[112]:
          Index = 124
          Value = 6.16
          Unit = Nm
          Description = dC1
        Row[113]:
          Index = 125
          Value = 6.16
          Unit = Nm
          Description = dC2
        Row[114]:
          Index = 126
          Value = 6.16
          Unit = Nm
          Description = dC3
      DynamicLimits = DynParTables
        GearboxLimitsTableRef
        CrossSectionLimitsTableRef
      InternalDynamicLimits = Used
        TypeIsReadOnly = 1
        Type = D4-1100-S026
        GearboxLimits:
          Row[1]:
            Index = 0
            Value = 3
            Unit = 
            Description = Type of robot dyn par model
          Row[2]:
            Index = 1
            Value = 84.42
            Unit = Nm
            Description = Gearbox Drive 1
          Row[3]:
            Index = 2
            Value = 84.42
            Unit = Nm
            Description = Gearbox Drive 2
          Row[4]:
            Index = 3
            Value = 84.42
            Unit = Nm
            Description = Gearbox Drive 3
        CrossSectionLimits:
          Row[1]:
            Index = 0
            Value = 3
            Unit = Variant
            Description = 
          Row[2]:
            Index = 1
            Value = 10000
            Unit = N
            Description = 
          Row[3]:
            Index = 2
            Value = 10000
            Unit = N
            Description = 
          Row[4]:
            Index = 3
            Value = 10000
            Unit = N
            Description = 
          Row[5]:
            Index = 4
            Value = 10000
            Unit = Nm
            Description = 
          Row[6]:
            Index = 5
            Value = 10000
            Unit = Nm
            Description = 
          Row[7]:
            Index = 6
            Value = 10000
            Unit = Nm
            Description = 
          Row[8]:
            Index = 7
            Value = 225
            Unit = N
            Description = 
          Row[9]:
            Index = 8
            Value = 225
            Unit = N
            Description = 
          Row[10]:
            Index = 9
            Value = 225
            Unit = N
            Description = 
          Row[11]:
            Index = 10
            Value = 225
            Unit = N
            Description = 
          Row[12]:
            Index = 11
            Value = 225
            Unit = N
            Description = 
          Row[13]:
            Index = 12
            Value = 225
            Unit = N
            Description = 
      LoadDependentJerkLimitsIsReadOnly = 0
      LoadDependentJerkLimits = PayloadDependentJerkReduction
        JerkReduction[1]:
          PayloadInKgIsReadOnly = 0
          PayloadInKg = 0
          JerkReductionInPercentIsReadOnly = 0
          JerkReductionInPercent = 0
        JerkReduction[2]:
          PayloadInKgIsReadOnly = 0
          PayloadInKg = 0.35
          JerkReductionInPercentIsReadOnly = 0
          JerkReductionInPercent = 0
        JerkReduction[3]:
          PayloadInKgIsReadOnly = 0
          PayloadInKg = 1
          JerkReductionInPercentIsReadOnly = 0
          JerkReductionInPercent = 50
        JerkReduction[4]:
          PayloadInKgIsReadOnly = 0
          PayloadInKg = 1.5
          JerkReductionInPercentIsReadOnly = 0
          JerkReductionInPercent = 50
        JerkReduction[5]:
          PayloadInKgIsReadOnly = 0
          PayloadInKg = 3
          JerkReductionInPercentIsReadOnly = 0
          JerkReductionInPercent = 70
      CouplingsIsInvisible = 0
      JointAxesPositionLimits:
        JointAxisIsReadOnly = 0
        JointAxis[1] = UseAxisLimits
        JointAxis[2] = UseAxisLimits
        JointAxis[3] = UseAxisLimits
```

### Config_5.axesgroupfeature - 5APC3100_KBU3_000/mappMotion/Codian_D4r1100_1/Config_5.axesgroupfeature
```
Element Feature_Programs_D4r1100_1 (Type=axesgroupfeature)
  Type:
    InitialSettings:
      AccuracyHoldDelays = User defined
        UserAxesDelay = 0.065
    Location = User
      UserLocation[1]:
        FileDevice = CNC_Prg
```

### ComRobot.axesgroupfeature - 5APC3100_KBU3_000/mappMotion/ComRobot.axesgroupfeature
```
Element Feature_TrackingRobot (Type=axesgroupfeature)
  Type = Tracking
    MotionBehaviour:
      OutOfWorkspaceSynchronisation:
        Clearance = 10
      OutOfWorkspaceSychronized = AdjustedVelocity
        Clearance = 10
Element Feature_MFunctions (Type=axesgroupfeature)
  Type = MFunctions
    MFunction[1]:
      IndexType:
        Index = 16
      Blocking = Disabled
      InSimulation = Set
      PvMapping = ::APP_Robot1:M16
    MFunction[2]:
      IndexType:
        Index = 17
      Blocking = Disabled
      InSimulation = Set
      PvMapping = ::APP_Robot1:M17
    MFunction[3]:
      IndexType:
        Index = 32
      Blocking = Disabled
      InSimulation = Set
      PvMapping = ::APP_Robot1:M32
    MFunction[4]:
      IndexType:
        Index = 33
      Blocking = Disabled
      InSimulation = Set
      PvMapping = ::APP_Robot1:M33
    MFunction[5]:
      IndexType:
        Index = 34
      Blocking = Disabled
      InSimulation = Set
      PvMapping = ::APP_Robot1:M34
    MFunction[6]:
      IndexType:
        Index = 40
      Blocking = Disabled
      InSimulation = Set
      PvMapping = ::APP_Robot1:M40
Element Feature_PathDefRobot (Type=axesgroupfeature)
  Type = PathDefinitions
    PathDefinition[1]:
      Type:
        CalculatedIn = PCS
Element Feature_FrameHierachy (Type=axesgroupfeature)
  Type = FrameHierarchy
    FrameHierarchy = Custom
      FramePropertyMapping:
        BCS = RobotBase
      MCS:
        Frame[1]:
          Name = RobotBase
          Type:
            Translation:
              Z = 950
        Frame[2]:
          Name = UserFrame1
          Frame[1]:
            Name = FixedPlace
            Type:
              Translation:
                Y = 450
Element Feature_WorkspaceMonitoring (Type=axesgroupfeature)
  Type = WorkspaceMonitoring
    WorkspaceRef = Workspace_1
Element Feature_Selection (Type=axesgroupfeature)
  Type = TrackingFrameSelection
    Selectors:
      Selector[1]:
        Name = Infeed
        Filters:
          Filter[1]:
            TrackingPathRef[1] = gTrackingPathConveyor_1
          Filter[2] = SelectionArea
            Area[1]:
              Translation:
                X = -1500
                Y = -500
                Z = -1000
              Dimensions:
                Length = 1300
                Width = 1000
                Height = 1000
          Filter[3] = AttributeMask
            Mask = 2#00000000000000000000000000000001
      Selector[2]:
        Name = Outfeed
        Filters:
          Filter[1]:
            TrackingPathRef[1] = gTrackingPathConveyor_2
          Filter[2] = SelectionArea
            Area[1]:
              Translation:
                X = 0
                Y = -500
                Z = -1000
              Dimensions:
                Length = 1500
                Width = 1000
                Height = 1000
Element Feature_Programs (Type=axesgroupfeature)
  Type:
    DefaultLanguage = ST
```

### Config.mappmotioncfg - 5APC3100_KBU3_000/mappMotion/Config.mappmotioncfg
```
Element MappMotionConfiguration (Type=mappmotioncfg)
  Processing:
    SymmetricMultiprocessing = Used
  Diagnostics:
    Snapshot = NotUsed
```

### AxisAx_1.axis - 5APC3100_KBU3_000/mappMotion/Conveyor/AxisAx_1.axis
```
Element gAxis_Conveyor_2 (Type=axis)
  BaseType = LinearPeriodic
    PeriodSettings:
      Period = 100000.0
  MovementLimits = InternalForPathControlledAxis
    Position:
      LowerLimit = -8388608.0
      UpperLimit = 8388607.0
Element gAxis_Conveyor_1 (Type=axis)
  BaseType = LinearPeriodic
    PeriodSettings:
      Period = 100000.0
  MovementLimits = InternalForPathControlledAxis
    Position:
      LowerLimit = -8388608.0
      UpperLimit = 8388607.0
```

### Config_1.trackingpath - 5APC3100_KBU3_000/mappMotion/Conveyor/Config_1.trackingpath
```
Element gTrackingPathConveyor_2 (Type=trackingpath)  // Tracking Path with moving objects
  Type:
    MotionSource = Axis
      AxisRef = gAxis_Conveyor_2
    TrackingFrames:
      AutomaticDeletion:
        Condition[1]:
          MinPosition = -100
          MaxPosition = 3000
  SceneViewerObject:
    VisualRepresentation = Conveyor belt
      Dimensions:
        Length = 3000
        Width = 300
        Height = 1
      Translation:
        Y = -150
        Z = -50
Element gTrackingPathConveyor_1 (Type=trackingpath)  // Tracking Path with moving objects
  Type:
    MotionSource = Axis
      AxisRef = gAxis_Conveyor_1
    TrackingFrames:
      AutomaticDeletion:
        Condition[1]:
          MinPosition = -100
          MaxPosition = 3000
        Condition[2] = AfterDesynchronization
          AxesGroupRef = gAxesGroup_D4r1100_1
  SceneViewerObject:
    VisualRepresentation = Conveyor belt
      Dimensions:
        Length = 3000
        Width = 300
        Height = 1
      Translation:
        Y = -150
        Z = -50
```

### Config_7.axisfeature - 5APC3100_KBU3_000/mappMotion/Conveyor/Config_7.axisfeature
```
Element Feature_1 (Type=axisfeature)
  Type = ProfGen
    JerkFilter = JerkLimited
```

### Config_7.purevaxcfg - 5APC3100_KBU3_000/mappMotion/Conveyor/Config_7.purevaxcfg
```
Element PureVAxCfg_1 (Type=purevaxcfg)
  PureVAxis:
    AxisReference = gAxis_Conveyor_1
Element PureVAxCfg_2 (Type=purevaxcfg)
  PureVAxis:
    AxisReference = gAxis_Conveyor_2
```

## Logical view

Binary libraries used (declarations not repeated): operator, runtime, astime, AsIecCon, standard, AsBrStr, sys_lib, AsArSdm, brsystem, FileIO, AsIODiag, DataObj, AsArProf, AsMem, AsIOAcc, AsEPL, ASMcDcs, AsBrMath, visapi, ArTextSys, AsSem, AsZip, AcpInvLib 3.00.4, MpRecipe 6.0.0, MpUserX 6.0.0, MpFile 6.0.0, MpAlarmX 6.0.0, MpCom 6.0.0, CoTrace, MpServer, MpBase, McBase 6.4.0, McAxGroup 6.4.0, McAcpAx 6.4.0, McAxis 6.4.0, McPathGen 6.4.0, McTrkPath 6.4.0, MpAxis 6.4.0, McProgInt 6.4.0, McPureVAx 6.4.0, McDS402Ax 6.4.0, MpRobotics 6.4.0, MpCnc 6.4.0

### Global.typ
```iecst
TYPE
	ControlPanelInputs : 	STRUCT  (*Command Buttons*)
		StartSorting : BOOL; (*Run a sorting program*)
		StartPrePalletizing : BOOL; (*Run a pre palleticing application demo*)
		StartPickNPlace : BOOL; (*Run a pick and place application demo*)
		StartPlaceWithConditionalStop : BOOL; (*Rund a place position with conditional stop*)
		StartMultipickRandom : BOOL; (*Random product creation with multipick*)
		StartMultipick : BOOL; (*Rund a multipick application demo*)
		Reset : BOOL; (*Stop Execute*)
		VelocityProduction : REAL; (*Velocity for production [ppm]*)
		ProductGap : REAL; (*Length of the product [mm]*)
	END_STRUCT;
	ControlPanelType : 	STRUCT  (*Control Panel*)
		Input : ControlPanelInputs; (*Buttons *)
	END_STRUCT;
END_TYPE
```


### Package Logical/Conveyor - Device: 1 axis positioner

### Conveyor.typ
```iecst
TYPE
	ConveyorStatesEnum :
		( (*State of the robot*)
		STATE_INIT,
		STATE_WAIT,
		STATE_RESET,
		STATE_PRODUCTION,
		STATE_ERROR
		);
END_TYPE
```

### Program Logical/Conveyor/APP_Conveyor1 (IEC) - Motion Belt

#### Variables.var - Local variables
```iecst
(*
MpAxisBasic function blocks used for Conveyor Handling*)
VAR
	MpAxConveyor : MpAxisBasic;
	AxParConveyor : MpAxisBasicParType;
	Period : LREAL;
	LinkTrackingPath : UDINT;
	LinkAxis : UDINT;
END_VAR
(*
MpAxisBasicConfig function blocks*)
VAR
	LastProductPosition : LREAL := 0;
	State : ConveyorStatesEnum;
	Reset : BOOL;
	Start : BOOL;
	SetVelocity : REAL;
	ProductGap : LREAL;
	Multipick : BOOL;
END_VAR
(*
Tracking function*)
VAR
	MC_BR_TrackingFrameDelete_0 : MC_BR_TrackingFrameDelete;
	MC_BR_TrackingFrameCreate_0 : MC_BR_TrackingFrameCreate;
	createCnt : USINT;
	RandomCreation : BOOL;
END_VAR
```

#### Init.st - Init code
```iecst
PROGRAM _INIT

	DefineLinks;

	// Set Default Parameters of the Tracking Frames
	MC_BR_TrackingFrameCreate_0.Parameters.Attribute	:= 0;
	MC_BR_TrackingFrameCreate_0.Parameters.Translation.X := 0.0;
	MC_BR_TrackingFrameCreate_0.Parameters.Translation.Y := 0.0;
	MC_BR_TrackingFrameCreate_0.Parameters.Translation.Z := 0.0;
	MC_BR_TrackingFrameCreate_0.Parameters.Orientation.Angle1 := 0.0;
	MC_BR_TrackingFrameCreate_0.Parameters.Orientation.Angle2 := 0.0;
	MC_BR_TrackingFrameCreate_0.Parameters.Orientation.Angle3 := 0.0;
	MC_BR_TrackingFrameCreate_0.Parameters.Orientation.Type := 0;

	MC_BR_TrackingFrameDelete_0.Mode :=  mcTRKFRM_DELETE_MOD_ALL;

END_PROGRAM
```
